(****************************************************************************************)
(*							  Check for valid logical axis no.							*)
(****************************************************************************************)
IF NOT bIsChannelSpecific AND NOT HLI3_CheckAxisValid(nHliAxisIdx := nHliAxisIdx) THEN
	bError									:= TRUE;
	nErrorId								:= 10000;
	RETURN;
END_IF

IF NOT HLI3_CheckChannelValid(nChannel := nHliChannelIdx) THEN
	bError									:= TRUE;
	nErrorId								:= 20000;
	RETURN;	
END_IF

(****************************************************************************************)
(*											Reset										*)
(****************************************************************************************)
fbRtrigChannelReset
	(CLK := bChannelReset);

IF fbRtrigChannelReset.Q THEN
	nRevolution		:= 0;
	nPosition		:= 0;
	bAcknowledge	:= FALSE;
	M03				:= FALSE;
	M03_Internal	:= FALSE;
	M04				:= FALSE;
	M04_Internal	:= FALSE;
	M05				:= FALSE;
	M05_Internal	:= FALSE;
	M19				:= FALSE;
	M19_Internal	:= FALSE;	
	pM40^			:= FALSE;
	M40_Internal	:= FALSE;
	pM41^			:= FALSE;
	M41_Internal	:= FALSE;
	pM42^			:= FALSE;
	M42_Internal	:= FALSE;
	pM43^			:= FALSE;
	M43_Internal	:= FALSE;
	pM44^			:= FALSE;
	M44_Internal	:= FALSE;
	pM45^			:= FALSE;
	M45_Internal	:= FALSE;
END_IF

(****************************************************************************************)
(*									Receive requests from cnc							*)
(****************************************************************************************)
(* Look out for open technology function either on the channel or the axis specific		*)
(* section of the HLI, depending on parameter ''.										*)
IF bIsChannelSpecific THEN
	nOpenTechnoCount	:= gpCh[nHliChannelIdx]^.used_units_std_sync_r;
	nTechFctMaxidx 		:= gpCh[nHliChannelIdx]^.used_units_std_sync_r - 1;
ELSE
	nOpenTechnoCount	:= gpAx[nHliAxisIdx]^.used_units_std_sync_r;
	nTechFctMaxidx 		:= gpAx[nHliAxisIdx]^.used_units_std_sync_r - 1;
END_IF

IF nOpenTechnoCount > 0 THEN
	FOR nLoop := 0 TO nTechFctMaxIdx DO
		(* Depending on the source determined by parameter 'bIsChannelSpecific', the		*)
		(* channel or axis specific section of the HLI will be examined.					*)
		IF bIsChannelSpecific THEN
			pActTechnoUnit	:= ADR(gpCh[nHliChannelIdx]^.techno_unit_std_sync[nLoop]);
		ELSE
			(* Get current axis specifc technology data *)
			pActTechnoUnit	:= ADR(gpAx[nHliAxisIdx]^.techno_unit_std_sync[nLoop]);
		END_IF
	
		(* Check request *)
		IF pActTechnoUnit^.please_rw AND
		   NOT pActTechnoUnit^.done_w
		THEN
			CASE UINT_TO_UDINT(pActTechnoUnit^.fkt_ctrl_r) OF
		     (* -------------------------------------------------------------------------- *)
			 (* Handle M function *)
			 HLI_INTF_M_FKT:
				pMProcess					:= ADR(pActTechnoUnit^.attribut_r.data[0]);
				
				IF (pMProcess > 0) AND bHandleGearChange THEN
					CASE pMProcess^.nr OF
					 40:	M_ManageAcknowledgement(ADR(M40_Internal), pM40, ADR(bAcknowledge));
					 41:	M_ManageAcknowledgement(ADR(M41_Internal), pM41, ADR(bAcknowledge));
					 42:	M_ManageAcknowledgement(ADR(M42_Internal), pM42, ADR(bAcknowledge));
					 43:	M_ManageAcknowledgement(ADR(M43_Internal), pM43, ADR(bAcknowledge));
					 44:	M_ManageAcknowledgement(ADR(M44_Internal), pM44, ADR(bAcknowledge));
					 45:	M_ManageAcknowledgement(ADR(M45_Internal), pM45, ADR(bAcknowledge));
					END_CASE
				END_IF
				
			 (* -------------------------------------------------------------------------- *)
			 (* Handle S function *)
			 HLI_INTF_SPINDEL:
				pSProcess					:= ADR(pActTechnoUnit^.attribut_r.data[0]);
				
				(* If we are working with spindle functions provided by the channel 		*)
				(* specific section of the HLI the logical axis number transmitted from the *)
				(* CNC must fit the one given in parameter 'nLogAxisNoChannelSpecific'!					*)												
				IF bIsChannelSpecific AND (UINT_TO_INT(pSProcess^.log_achs_nr) <> nLogAxisNoChannelSpecific) THEN
					RETURN;
				END_IF
	
				CASE pSProcess^.move_cmd OF
				 (* ----------------------------------------------------------------------- *)
				 0: (* M19 *)
					IF (pSProcess^.pos_cmd = 19) AND
					   NOT M19_Internal THEN
						nPosition			:= pSProcess^.pos;
						M19_Internal		:= TRUE;
						M19					:= TRUE;
					ELSE
						IF NOT M19 THEN
							M19_Internal	:= FALSE;
							bAcknowledge	:= TRUE;
						END_IF
					END_IF
	
				 (* ----------------------------------------------------------------------- *)
				 3: (* M03 *)
					nRevolution				:= pSProcess^.rev;
	
					IF NOT M03_Internal THEN
						M03_Internal		:= TRUE;
						M03					:= TRUE;
					ELSE
						IF NOT M03 THEN
							M03_Internal	:= FALSE;
							bAcknowledge	:= TRUE;
						END_IF
					END_IF
	
				 (* ----------------------------------------------------------------------- *)
				 4: (* M04 *)
					nRevolution				:= pSProcess^.rev;
	
					IF NOT M04_Internal THEN
						M04_Internal		:= TRUE;
						M04					:= TRUE;
					ELSE
						IF NOT M04 THEN
							M04_Internal	:= FALSE;
							bAcknowledge	:= TRUE;
						END_IF
					END_IF
	
				 (* ----------------------------------------------------------------------- *)
				 5: (* M05 *)
					IF NOT M05_Internal THEN
						M05_Internal		:= TRUE;
						M05					:= TRUE;
					ELSE
						IF NOT M05 THEN
							M05_Internal	:= FALSE;
							bAcknowledge	:= TRUE;
						END_IF
					END_IF
	
				END_CASE
			END_CASE
	
			(* Handle acknowledgement *)
			IF bAcknowledge THEN
				bAcknowledge				:= FALSE;
				nRevolution					:= 0;
				nPosition					:= 0;
				pActTechnoUnit^.please_rw 	:= FALSE;
		   		pActTechnoUnit^.done_w		:= TRUE;
			END_IF
		END_IF
	END_FOR
	
END_IF
END_ACTION

{attribute 'object_name' := 'M_ManageAcknowledgement'}
METHOD PRIVATE M_ManageAcknowledgement
VAR_INPUT
	pInternal: POINTER TO BOOL;
	pPublic: POINTER TO BOOL;
	pAcknowledgement: POINTER TO BOOL;
END_VAR
IF NOT pInternal^ THEN
	pInternal^			:= TRUE;
	pPublic^			:= TRUE;	
ELSIF NOT pPublic^ THEN
	pInternal^			:= FALSE;
	pAcknowledgement^	:= TRUE;
END_IF
END_METHOD

END_FUNCTION_BLOCK

// ---- CNC Beckhoff/3 Control/HLI3_SetAxisOverride.TcPOU
FUNCTION HLI3_SetAxisOverride : BOOL
VAR_INPUT
	/// number of Axis 
	nHliAxisIdx: INT;
	nOverride: UINT;
END_VAR

(* ========================================================= *)
(*    FUN: HLI_SetAxisOverride                               *)
(* --------------------------------------------------------- *)
(*   Desc: Set the Axis Override                             *)
(* Author: TV                                                *)
(*   Date: 20.12.2007                                        *)
(*   Rev.: 1.0                                               *)
(*   Rev.: 1.1 MiB 19.11.2012 Tc3                            *)
(* ========================================================= *)
IF NOT (HLI3_CheckAxisValid(nHliAxisIdx := nHliAxisIdx)) THEN
	HLI3_SetAxisOverride := FALSE;
	RETURN;
END_IF


(* Limit the override *)
IF nOverride > 1200	THEN nOverride := 1200; END_IF
IF nOverride < 0 THEN nOverride := 0; END_IF

	gpAx[nHliAxisIdx]^.ipo_mc_control.override.enable_w  := TRUE;
	gpAx[nHliAxisIdx]^.ipo_mc_control.override.command_w := nOverride;

HLI3_SetAxisOverride := TRUE;

END_FUNCTION

// ---- CNC Beckhoff/PRG_ManualMode.TcPOU
PROGRAM PRG_ManualMode
VAR
	
END_VAR

(****************************************************************************************)
(* POU:		PRG_ManualMode                      										*)
(* Type:	PRG																			*)
(* Author: 	HR                                               							*)
(* Date: 	24.01.11																	*)
(* Rev.: 	1.0                                               							*)
(* ------------------------------------------------------------------------------------ *)
(* Desc:	Calls the appropriate manual mode handler									*)
(****************************************************************************************)

(* By default 'geManualModeController' is 'HMI'. Therefore program 'PRG_ManualModeHMI'	*)
(* is called in order to map manual mode signals from HMI to the manual mode control	*)
(* structures. By changing 'geManualModeController´s' value one can call different sub	*)
(* programs to set them in a application specific way.
									*)
geManualModeController := HMI;


CASE geManualModeController OF
	HMI:		PRG_ManualModeHMI();
	PANEL:		;
	REMOTE:		;
	CUSTOMER:	;
END_CASE

END_PROGRAM

// ---- CNC Beckhoff/PRG_ManualModeHMI.TcPOU
PROGRAM PRG_ManualModeHMI
VAR
	fbUintUdInt: ARRAY [0..MAX_USED_CHANNEL_IDX] OF FB_Uint_Udint;
	nHandwheel : UINT;		(* increments for handwheel (e.g. EL5101   *)
	nHandWheelBig: UDINT;
	i: INT;
END_VAR


FOR i := 0 TO MAX_USED_CHANNEL_IDX DO
	
	IF (HLI3_CheckChannelValid(i)) THEN

		stManualModeParameter[i].stChannelParameter.nChanIdx						:= i;       (* Channel 1 *)
		stManualModeParameter[i].stChannelParameter.nInc							:= PLCMachineMode[i+1].ManualMode.nInc * 10;
		
		stManualModeParameter[i].stChannelParameter.eManualType						:= UINT_TO_INT(PLCMachineMode[i+1].ManualMode.nManualTyp);			
		IF (stManualModeParameter[i].stChannelParameter.eManualType = E_CNC_ManualType.Handwheel AND i <> PLCSelectedChannel-1) THEN	(* if in Handwheel mode and the channel is NOT selected -> leave handwheel mode and change to TippMode*)
			stManualModeParameter[i].stChannelParameter.eManualType						:= E_CNC_ManualType.TippMode;
		END_IF		
		
		stManualModeParameter[i].stChannelParameter.nHandwheelResolution			:= UDINT_TO_DINT(PLCMachineMode[i+1].ManualMode.nHwResolution);    (* 0.1 µm /rev (from HMI) *)						
		stManualModeParameter[i].stAxisParameter.stControlUnit[0].nLogAxisNr		:= PLCMachineMode[i+1].ManualMode.nLogAxisNumber;   (* Log. Achs Nummer *)
		IF stManualModeParameter[i].stAxisParameter.stControlUnit[0].nLogAxisNr = 0 THEN
			stManualModeParameter[i].stAxisParameter.stControlUnit[0].nLogAxisNr := gpCh[i]^.bahn_state.coord_r[0].log_achs_nr_r;
			PLCMachineMode[i+1].ManualMode.nLogAxisNumber := gpCh[i]^.bahn_state.coord_r[0].log_achs_nr_r;
		END_IF
		stManualModeParameter[i].stAxisParameter.stControlUnit[0].nSpeed			:= LREAL_TO_UDINT(PLCMachineMode[i+1].ManualMode.nSpeed * 16.666);
		stManualModeControlElements[i].stControlKeys[0].bKeyNeg						:= PLCMachineMode[i+1].ManualMode.bKeyNeg;
		stManualModeControlElements[i].stControlKeys[0].bKeyPos						:= PLCMachineMode[i+1].ManualMode.bKeyPos;
		stManualModeControlElements[i].stControlKeys[0].bKeyRapid					:= PLCMachineMode[i+1].ManualMode.bKeyRapid;
		
		(* the cnc needs an UDINT for handwheel increments, fbUintUdint extends an UInt to an UDINT *)
		(* the resoltion of the handwheel is parameterized in CNC-Task GEO/Manual MDS: (e.g. 400 handwheel inc / handwheel revolution
		
				hr_data[0].hr_aufl_z              400         ( P-MANU-00005 : Handwheel resolution numerator
				hr_data[0].hr_aufl_n                1     	  ( P-MANU-00006 : Handwheel resolution denominator
		*) 
		fbUintUdInt[i](nInSmall := nHandwheel, nBig := nHandWheelBig);
		stManualModeControlElements[i].nHandwheelInc[0] :=  UDINT_TO_DINT(nHandWheelBig);
  END_IF
END_FOR

END_PROGRAM

// ---- CNC Beckhoff/Util/FB_Uint_Udint.TcPOU
FUNCTION_BLOCK FB_Uint_Udint
VAR
	nOldValue: UINT;
	nDiff: DINT;
	nMinus: BOOL;
	nPlus: BOOL;
END_VAR
VAR_INPUT
	nInSmall: UINT;
END_VAR

VAR_IN_OUT
	nBig: UDINT;
END_VAR

nDiff := nInSmall - nOldValue;


(* Richtung Minus *)
IF ndiff > 10000 THEN
	nBig := nBig - 1;
	nMinus := TRUE;
END_IF

(* Richtung Plus *)
IF ndiff < -10000 THEN
	nBig := nBig + 1;
	nPlus := TRUE;
END_IF

IF (ndiff < 500) AND ndiff > -500 THEN
  nBig := DINT_TO_UDINT( UDINT_TO_DINT(nBig) + nDiff) ;
END_IF
nOldValue := nInSmall;

END_FUNCTION_BLOCK

// ---- CNC Beckhoff/PRG_ChannelHandler.TcPOU
PROGRAM PRG_ChannelHandler
VAR	
	nChan					: INT;
	nOldSelectedChannel		: UDINT;
	CNCChannel				: ARRAY[0..MAX_USED_CHANNEL_IDX] OF HLI3_CNCChannel;	
	BlockSearch_Channel		: ARRAY[0..MAX_USED_CHANNEL_IDX] OF HLI3_BlockSearch;
	ModeManual_Channel		: ARRAY[0..MAX_USED_CHANNEL_IDX] OF HLI3_ManualModeHandler;
	ErrorHandler_Channel	: ARRAY[0..MAX_USED_CHANNEL_IDX] OF FB_ChannelError;
	nChanNo: UDINT;	
	i: INT;
	
END_VAR

(****************************************************************************************)
(* POU:		PRG_ChannelHandler                     										*)
(* Type:	PRG																			*)
(* Author: 	HR / TV / MiB                                          						*)
(* Date: 	23.01.11																	*)
(* Last:	02.03.16																	*)
(* Rev.: 	1.4                                              							*)
(* ------------------------------------------------------------------------------------ *)
(* Desc:	Description																	*)
(****************************************************************************************)

(****************************************************************************************)
(*	  Map CNC function selection from HMI to selected channel (and state vice versa)  	*)
(****************************************************************************************)
IF (nOldSelectedChannel <>INT_TO_UDINT(PLCSelectedChannel)) THEN
	PLCChannelSignals.SingleBlock 		:= PLCMachineMode[PLCSelectedChannel].ChannelSignals.SingleBlock;
	PLCChannelSignals.PrgBlockIgnore	:= PLCMachineMode[PLCSelectedChannel].ChannelSignals.PrgBlockIgnore;
	PLCChannelSignals.M01Stop 			:= PLCMachineMode[PLCSelectedChannel].ChannelSignals.M01Stop;
	PLCChannelSignals.Backward 			:= PLCMachineMode[PLCSelectedChannel].ChannelSignals.Backward;
	PLCChannelSignals.FeedHold 			:= PLCMachineMode[PLCSelectedChannel].ChannelSignals.FeedHold;
	nOldSelectedChannel 				:= INT_TO_UDINT(PLCSelectedChannel);
END_IF

PLCMachineMode[PLCSelectedChannel].ChannelSignals.SingleBlock 		:= PLCChannelSignals.SingleBlock;
PLCMachineMode[PLCSelectedChannel].ChannelSignals.PrgBlockIgnore 	:= PLCChannelSignals.PrgBlockIgnore;
PLCMachineMode[PLCSelectedChannel].ChannelSignals.M01Stop 			:= PLCChannelSignals.M01Stop;
PLCMachineMode[PLCSelectedChannel].ChannelSignals.Backward 		:= PLCChannelSignals.Backward;
PLCMachineMode[PLCSelectedChannel].ChannelSignals.FeedHold 		:= PLCChannelSignals.FeedHold;



FOR i := 0 TO MAX_USED_CHANNEL_IDX DO
		
	nChan := i;	
	IF (HLI3_CheckChannelValid(nChan)) THEN		
		
		(* Error handler for channel 1 *)
		ErrorHandler_Channel[nChan](nChanIdx			:= nCHan);
		
		(* Pass feedrate override from HMI to first channel (in [0.1%]) *)
		HLI3_SetChannelOverride
			(nChanIdx			:= nChan,
			 nOverride			:= PLCFeedOverride * 10
			);
		
		(* Channel interface *)
		CNCChannel[nChan]
			(nChanIdx			:= nChan,
			 (* Operation Mode *)
			 bModeStandby		:= PLCMachineMode[nChan+1].Standby,
			 bModeAutomatic		:= PLCMachineMode[nChan+1].Automatic,
			 bModeManual		:= PLCMachineMode[nChan+1].Manual,
			 bModeMDI			:= PLCMachineMode[nChan+1].MDI,	 
			 bModeReference		:= PLCMachineMode[nChan+1].Homing,
			 (* Operation State *)
			 bStateSelect		:= PLCMachineMode[nChan+1].Select,
			 bStateReady		:= PLCMachineMode[nChan+1].Ready,
			 bStateStart		:= PLCMachineMode[nChan+1].Start,
			 bStateStop			:= PLCMachineMode[nChan+1].Stop,
			 bStateReset		:= PLCMachineMode[nChan+1].Reset,
			 (* Special Functions *)
			 sProgramName		:= PLCMachineMode[nChan+1].ProgramName,
			 sMDIString			:= PLCMachineMode[nChan+1].MDIString,
			 bBackwardMotion	:= PLCMachineMode[nChan+1].ChannelSignals.Backward,
			 bPrgBlockIgnore	:= PLCMachineMode[nChan+1].ChannelSignals.PrgBlockIgnore,
			 bFeedHold			:= PLCMachineMode[nChan+1].ChannelSignals.FeedHold,
			 bSingleBlock		:= PLCMachineMode[nChan+1].ChannelSignals.SingleBlock,
			 bDoSingleBlock		:= PLCMachineMode[nChan+1].ChannelSignals.DoSingleBlock,
			 bM01Stop			:= PLCMachineMode[nChan+1].ChannelSignals.M01Stop,
			 nSyntaxCheck		:= PLCMachineMode[nChan+1].SyntaxCheck.nType,
			 sManualInitString  :=  stManualModeParameter[nChan].stChannelParameter.strInitParameter
			);
		
		(* Handle block search *)
		BlockSearch_Channel[nChan]
			(nChanIdx			:= nChan,
			 bStartRead      	:= PLCMachineMode[nChan+1].BlockSearch.bStartRead,   (* Edge signal *)
			 bStartWrite     	:= PLCMachineMode[nChan+1].BlockSearch.bStartWrite,  (* Edge signal *)
			 BlockSearch		:= PLCMachineMode[nChan+1].BlockSearch
			);
		
		CNCSystem.Channel[nChan].ActDistance 	:= DINT_TO_LREAL(BlockSearch_Channel[nChan].coveredDistance_AfterReset) / 10.0;
		CNCSystem.Channel[nChan].ActBlockCount 	:= BlockSearch_Channel[nChan].actualBlockCount_AfterReset;
		
		
		ModeManual_Channel[nChan]
			(stManualModeParameter  	 	:= stManualModeParameter[nChan],
			 stManualModeControlElements	:= stManualModeControlElements[nChan],
			 stManualModeControlElementState := stManualModeControlElementState,
			 bReset 						:= FALSE,
			 arrAxisInG201 				=> stManualModeState[nChan].arrAxisInG201
			);
	END_IF
END_FOR

END_PROGRAM

// ---- CNC Beckhoff/2 OperationMode/HLI3_CNCChannel.TcPOU
FUNCTION_BLOCK HLI3_CNCChannel
VAR_INPUT
	/// index of channel 
	nChanIdx: INT;
	/// must be xxx.nc 
	sProgramName: STRING(HLI_IMCM_MODE_STATE_PARAM_STRL);
	/// the MDI string 
	sMDIString: STRING(HLI_IMCM_MODE_STATE_PARAM_STRL);
	/// static signal 
	bBackwardMotion: BOOL;
	/// static signal 
	bFeedHold: BOOL;
	/// static signal 
	bReducedFeed: BOOL;
	/// static signal 
	bSingleBlock: BOOL;
	/// static signal 
	bPrgBlockIgnore: BOOL;
	/// static signal 
	bM01Stop: BOOL;
	/// static signal 
	nSyntaxCheck: DINT;
	/// initi parameter for manual mode
	sManualInitString	     : STRING;
END_VAR
VAR_IN_OUT
	/// please only a flank 
	bModeStandby: BOOL;
	/// please only a flank 
	bModeAutomatic: BOOL;
	/// please only a flank 
	bModeManual: BOOL;
	/// please only a flank 
	bModeMDI: BOOL;
	/// please only a flank 
	bModeReference: BOOL;
	/// please only a flank 
	bStateSelect: BOOL;
	/// please only a flank 
	bStateReady: BOOL;
	/// please only a flank 
	bStateStart: BOOL;
	/// please only a flank 
	bStateStop: BOOL;
	/// please only a flank 
	bStateReset: BOOL;
	/// please only a flank 
	bDoSingleBlock: BOOL;
END_VAR
VAR
	bGoToActive	: BOOL;
	/// Pointer to HLI Motion Control Unit 
	pUnit: POINTER TO MC_CONTROL_MCM_MODE_STATE_UNIT;
	/// Pointer to HLI channel command 
	pCommand: POINTER TO HLI_PROC_TRANS_TO_MODE_STATE;
	/// Pointer to channel control structure 
	pChannel: POINTER TO ST_CncChannel;
	ChannelMHTFunction: HLI3_QuitChannelMHTFunction;
	/// Current Mode of Operation Modes;
	currentMode: UDINT;
	/// Current State of Operation Modes;
	currentState: UDINT;
	idx: INT;
	bEndOfManualMode: BOOL;
	bCheckOpModeFirst: BOOL;
	fbRTrigReset: R_TRIG;
	bResetRequest: BOOL;
	ChannelResetRequest: HLI3_ChannelResetRequest;
	nChan: INT;
	nStateAutoMDIStart: INT;
END_VAR

(* ========================================================= *)
(*     FB: HLI_CNCChannel                                    *)
(* --------------------------------------------------------- *)
(*   Desc:                                                   *)
(*   Author: MK ,MiB, TV, Rch                                *)
(*   Date: 2017.05.08                                        *)
(*   Rev.: 1.6                                               *)
(*         1.2 Before "start" the state is swicthed to 		 *)
(*				"Selected" and "Ready" to ensure that the    *)	
(*				actual selected program will start 			 *)
(*		   1.3  BugFix : nChanNo at HLI3_ChannelModeMDI()    *)
(*         1.4  Implement state switch to "selected" and "ready"  *)         
(*		   1.5  Channel reset via commanding state 			 *)
(*              RESETTING directly							 *)  
(*		   1.6  Optimized Channel reset via commanding state *)
(*				RESETTING directly						     *)
(*		   1.7  Init Paramerer for Manual mode as input parameter*)
(* ========================================================= *)

IF NOT HLI3_CheckChannelValid(nChannel := nChanIdx) THEN
	RETURN;
END_IF


(* handle reset request *)
fbRTrigReset
	(CLK := bStateReset);
	
IF fbRTrigReset.Q THEN
	nStateAutoMDIStart := 0;
END_IF

(* set up pointer *)
pUnit    := ADR(gpCh[nChanIdx]^.channel_mc_control.mode_and_state);
pCommand := ADR(pUnit^.command_w);


(* ************************************* *)
(*  Motion-Control                       *)
(* ************************************* *)
(* Backward Motion *)
HLI3_ChannelSetBackwardMotion(nChanIdx:=nChanIdx, bBackwardMotion:=bBackwardMotion);

(* Program Block Ignore *)
HLI3_ChannelSetProgramBlockIgnore(nChanIdx:=nChanIdx, bPrgBlockIgnore:=bPrgBlockIgnore);

(* Feed Hold *)
HLI3_ChannelSetFeedHold(nChanIdx:=nChanIdx, bFeedHold:=bFeedHold);

(* Single Step *)
HLI3_ChannelSetSingleBlock(nChanIdx:=nChanIdx, bSingleBlock:=bSingleBlock);

(* Reduced Feed *)
HLI3_ChannelSetReducedFeed(nChanIdx:=nChanIdx, bReducedFeed:=bReducedFeed);

(* Syntax Check *)
gpCh[nChanIdx]^.decoder_mc_control.execution_mode.command_w := nSyntaxCheck;

(* Optional stop M01 *)
gpCh[nChanIdx]^.bahn_mc_control.m01_stop_enable.command_w := bM01Stop;


(* ************************************ *)
(*  MHT-Function                        *)
(* ************************************ *)
(* Reset all M- and H-Functions whenn 	*)
(* the channel gets resetted			*)
IF (pChannel > 0) THEN
	IF (pChannel^.ActState = HLI_IMCM_PROCESS_RESETTING) THEN
		HLI3_ChannelResetMFunctions(nChanIdx);
		HLI3_ChannelResetHFunctions(nChanIdx);
	END_IF
END_IF

(* MHT-Function, channel *)
ChannelMHTFunction(nChanIdx:=nChanIdx);

(* ************************************* *)
(*  Channel Status Info and error        *)
(* ************************************* *)
HLI3_GetChannelStatusInfo(nChanIdx:=nChanIdx);
HLI3_GetChannelError(nChanIdx:=nChanIdx);

(* ************************************* *)
(*  do single stepping                   *)
(* ************************************* *)
(* Achtung: hier noch anpassen, nur in Abhaengigkeit vom aktuellen Status den Start setzen *)
IF bDoSingleBlock THEN
	bDoSingleBlock := FALSE;
	bStateStart 	:= TRUE;
END_IF

(* ************************************* *)
(*  Operation Modes                      *)
(* ************************************* *)
(* Target modes and states *)
pChannel := ADR(CNCSystem.Channel[nChanIdx]);
OpModes();

(* OperationMode Standby *)
IF pChannel^.Mode.Standby = TRUE THEN
	HLI3_ChannelModeStandby(ProgramName:=sProgramName, pUnit:=pUnit, pCommand:=pCommand, pChannel:=pChannel);
END_IF

(* OperationMode Auto *)
IF pChannel^.Mode.Auto = TRUE THEN
	HLI3_ChannelModeAuto(ProgramName:=sProgramName, pUnit:=pUnit, pCommand:=pCommand, pChannel:=pChannel);
END_IF

(* OperationMode MDI *)
IF pChannel^.Mode.MDI THEN
	(*sProgramName := PLCCncMDIString;*)
	HLI3_ChannelModeMDI(pMDIString:=ADR(sMDIString), pUnit:=pUnit, pCommand:=pCommand, pChannel:=pChannel);
END_IF

(* OperationMode Reference *)
//IF pChannel^.Mode.REFERENCE THEN TC3HR
IF pChannel^.Mode.Homing THEN
	sProgramName := '';	(* we choose the default program: rpf.nc *)
	HLI3_ChannelModeReference(sRefPosString:=sProgramName, pUnit:=pUnit, pCommand:=pCommand, pChannel:=pChannel);
END_IF

(* OperationMode Manual *)
IF pChannel^.Mode.Manual THEN
	bEndOfManualMode := FALSE;
	HLI3_ChannelModeManual(pUnit:=pUnit, pCommand:=pCommand, pChannel:=pChannel, sManualInitString := sManualInitString);
END_IF

(* end of manual mode *)
IF (pChannel^.Mode.Standby
OR pChannel^.Mode.Auto
OR pChannel^.Mode.MDI
//OR pChannel^.Mode.REFERENCE) THEN TC3HR
OR pChannel^.Mode.Homing) THEN
	bEndOfManualMode := TRUE;
END_IF

(* Reset *)
HLI3_ChannelReset(nChanIdx:=nChanIdx);							(* channel *)
FOR idx := 0 TO UDINT_TO_INT(gNrAx) DO							(* axis *)
	HLI3_AxisReset(nChanNo:=nChanIdx+1, nHliAxisIdx:=idx);
END_FOR

ACTION AutoMDIStart:



CASE nStateAutoMDIStart OF
	0:		;(* IDLE *)
	
	10: (* swicth to selected *)
		pChannel^.State.Selected := TRUE;
		nStateAutoMDIStart := nStateAutoMDIStart +10;
		
	20: (* wait for selected *)
		IF (pChannel^.ActState =  HLI_IMCM_PROCESS_SELECTED) THEN
			pChannel^.State.Ready := TRUE;
			nStateAutoMDIStart := nStateAutoMDIStart +10;
		END_IF
	30: (* Wait for ready and then start*)
		IF (pChannel^.ActState =  HLI_IMCM_PROCESS_READY) THEN
			pChannel^.State.Start := TRUE; 
			nStateAutoMDIStart := 0;
		END_IF
	
END_CASE
END_ACTION

ACTION OpModes:
(*************************************************)
(* Restore internal state at first run           *)
(* after PLC reset                               *)
(*************************************************)

IF bCheckOpModeFirst = FALSE THEN
	bCheckOpModeFirst := TRUE;
	currentMode := HLI3_GetChannelMode(nChanIdx:=nChanIdx);
	IF currentMode = HLI_IMCM_STANDBY_MODE THEN
		pChannel^.Mode.Standby := TRUE;
	END_IF
	IF currentMode = HLI_IMCM_AUTOMATIC_MODE THEN
		pChannel^.Mode.Auto := TRUE;
	END_IF
	IF currentMode = HLI_IMCM_MDI_MODE THEN
		pChannel^.Mode.MDI := TRUE;
	END_IF
	IF currentMode = HLI_IMCM_MANUAL_MODE THEN
		pChannel^.Mode.Manual := TRUE;
	END_IF
	IF currentMode = HLI_IMCM_REFERENCE_MODE THEN
		//pChannel^.Mode.REFERENCE := TRUE; TC3HR
		pChannel^.Mode.Homing := TRUE;
	END_IF
END_IF


(*************************************************)
(* Operation Modes                               *)
(*************************************************)

IF bModeStandby THEN
	bModeStandby := FALSE;
	pChannel^.Mode.Standby		:= TRUE;
	pChannel^.Mode.Auto			:= FALSE;
	pChannel^.Mode.MDI			:= FALSE;
	pChannel^.Mode.Manual		:= FALSE;
	pChannel^.Mode.Homing		:= FALSE;


	pChannel^.State.Selected	:= TRUE;
END_IF

IF bModeAutomatic THEN
	bModeAutomatic 				:= FALSE;
	bGoToActive					:= FALSE;
	pChannel^.Mode.Standby		:= FALSE;
	pChannel^.Mode.Auto			:= TRUE;
	pChannel^.Mode.MDI			:= FALSE;
	pChannel^.Mode.Manual		:= FALSE;
	pChannel^.Mode.Homing		:= FALSE;

	pChannel^.State.Selected	:= TRUE;
END_IF

IF bModeMDI THEN
	bModeMDI := FALSE;
	bGoToActive					:= FALSE;
	pChannel^.Mode.Standby		:= FALSE;
	pChannel^.Mode.Auto			:= FALSE;
	pChannel^.Mode.MDI			:= TRUE;
	pChannel^.Mode.Manual		:= FALSE;
	pChannel^.Mode.Homing		:= FALSE;

	pChannel^.State.Selected	:= TRUE;
END_IF

IF bModeManual THEN
	bModeManual := FALSE;
	pChannel^.Mode.Standby		:= FALSE;
	pChannel^.Mode.Auto			:= FALSE;
	pChannel^.Mode.MDI			:= FALSE;
	pChannel^.Mode.Manual		:= TRUE;
	pChannel^.Mode.Homing		:= FALSE;

	pChannel^.State.Start		:= TRUE;
END_IF

IF bModeReference THEN
	bModeReference := FALSE;
	bGoToActive					:= FALSE;
	pChannel^.Mode.Standby		:= FALSE;
	pChannel^.Mode.Auto			:= FALSE;
	pChannel^.Mode.MDI			:= FALSE;
	pChannel^.Mode.Manual		:= FALSE;
	pChannel^.Mode.Homing		:= TRUE;
	
	pChannel^.State.Start		:= TRUE;
END_IF



(*************************************************)
(* Operation States                              *)
(*************************************************)

currentMode := HLI3_GetChannelMode(nChanIdx:=nChanIdx);
currentState := HLI3_GetChannelState(nChanIdx:=nChanIdx);

CASE currentMode OF
	(*-------------------------------------------------------------------*)
	HLI_IMCM_STANDBY_MODE:
		IF bStateReset THEN
			pChannel^.Mode.Standby := TRUE;
			pChannel^.State.Reset := TRUE;
		END_IF

	(*-------------------------------------------------------------------*)
	HLI_IMCM_AUTOMATIC_MODE:
		IF bStateStart THEN  (* replaced a simple 'start' by a sequence which switches the state to selected and ready*)
			IF currentState <> HLI_IMCM_PROCESS_HOLD AND currentState <> HLI_IMCM_PROCESS_ACTIVE THEN
				nStateAutoMDIStart := 10;
			ELSE
				pChannel^.State.Start := TRUE; 
			END_IF					   	
		END_IF
		IF nStateAutoMDIStart <> 0 THEN
			AutoMDIStart();
		END_IF

		IF bStateStop AND currentState <> HLI_IMCM_PROCESS_DESELECTED THEN
			pChannel^.State.Stop := TRUE;
		END_IF

		IF bStateReady THEN
			pChannel^.State.Ready := TRUE;
		END_IF

		IF bStateReset THEN
			pChannel^.State.Reset := TRUE;
		END_IF
		
		IF bStateSelect THEN
			pChannel^.State.Selected := TRUE;
		END_IF		

	(*-------------------------------------------------------------------*)
	HLI_IMCM_MDI_MODE:
		IF bStateStart THEN
			IF currentState <> HLI_IMCM_PROCESS_HOLD AND currentState <> HLI_IMCM_PROCESS_ACTIVE THEN
				nStateAutoMDIStart := 10;
			ELSE
				pChannel^.State.Start := TRUE; 
			END_IF
		END_IF
		
		IF nStateAutoMDIStart <> 0 THEN
			AutoMDIStart();
		END_IF
		
		IF bStateStop AND currentState <> HLI_IMCM_PROCESS_DESELECTED THEN
			pChannel^.State.Stop := TRUE;
		END_IF

		IF bStateSelect THEN
			pChannel^.State.Selected := TRUE;
		END_IF
		
		IF bStateReady THEN
			pChannel^.State.Ready := TRUE;
		END_IF

		IF bStateReset THEN
			pChannel^.State.Reset := TRUE;
		END_IF

	(*-------------------------------------------------------------------*)
	HLI_IMCM_MANUAL_MODE:
		IF bStateStart OR ((currentState = HLI_IMCM_PROCESS_SELECTED) AND bGoToActive) THEN
			pChannel^.State.Start 	:= TRUE;
		END_IF

		IF bStateReady THEN
			pChannel^.State.Ready 	:= TRUE;
		END_IF

		IF bStateSelect THEN
			pChannel^.State.Selected := TRUE;
		END_IF

		IF bStateStop THEN
			pChannel^.State.Stop := TRUE;
		END_IF

		IF bStateReset THEN
			bGoToActive := TRUE;
			pChannel^.State.Reset := TRUE;
		END_IF

	(*-------------------------------------------------------------------*)
	HLI_IMCM_REFERENCE_MODE:
		IF bStateStart THEN
			pChannel^.State.Start := TRUE;
		END_IF

		IF bStateStop THEN
			pChannel^.State.Stop := TRUE;
		END_IF

		IF bStateReset THEN
			pChannel^.State.Reset := TRUE;
		END_IF
END_CASE


bStateStart 	:= FALSE;
bStateStop 		:= FALSE;
bStateReset 	:= FALSE;
bStateSelect 	:= FALSE;
bStateready 	:= FALSE;
END_ACTION

END_FUNCTION_BLOCK

// ---- CNC Beckhoff/4 MHT-Function/HLI3_QuitChannelMHTFunction.TcPOU
FUNCTION_BLOCK HLI3_QuitChannelMHTFunction
VAR_INPUT
	/// Number of channel 
	nChanIdx: INT;
END_VAR
VAR_OUTPUT
	bOK: BOOL;
END_VAR
VAR
	ChannelMFunction: HLI3_DoChannelMFunction;
	ChannelTFunction: HLI3_DoChannelTFunction;
	ChannelHFunction: HLI3_DoChannelHFunction;
	/// local pointer to Data of actual Channel 
	pChannelData: POINTER TO HIGH_LEVEL_INTERFACE_CH;
	/// local pointer to actual techno unit 
	pActTechnoUnit: POINTER TO TECHNO_UNIT_CH;
	/// Index of axis specific technology function at HLI 
	nTechFctMaxIdx: UINT;
	/// loop variable 
	idx: UINT;
	/// number of M-function 
	nFuncNr: UDINT;
	nArgument: DINT;
	/// basis id of a tool 
	nToolBasicId: UDINT;
	pMHProcess: POINTER TO HLI_M_H_PROZESS;
	pSProcess: POINTER TO HLI_S_PROZESS;
	pTProcess: POINTER TO HLI_T_PROZESS;
	stAttributeData: St_TechnoAttributeData;
END_VAR

(* ========================================================= *)
(*     FB: HLI3_QuitChannelMHTFunction                        *)
(* --------------------------------------------------------- *)
(*   Desc:                                                   *)
(* Author: MK                                                *)
(*   Rev.: 1.1                                               *)
(*   Date: 18.07.2002                                        *)
(*       : 08.04.2005                                        *)
(*          24.11.2010 MiB Erweiterung um H Funktionen 		 *)
(* ========================================================= *)
(* Rev.:	1.2												 *)
(* Date:	02.10.2010                                    	 *)
(* Author:	HR												 *)
(* Author:	Added support for additional m function number	 *)
(* ========================================================= *)
(* Rev.:	1.3												 *)
(* Date:	26.01.2011                                    	 *)
(* Author:	HR												 *)
(* Author:	Added support for additional h function number	 *)
(* ========================================================= *)
(* Rev.:	1.4												 *)
(* Date:	20.11.2012                                    	 *)
(* Author:	MiB												 *)
(* Author:	TC3												 *)
(* ========================================================= *)
(* Rev.:	1.4.1									         *)
(* Date:	15.07.2013                                    	 *)
(* Author:	TV												 *)
(* ========================================================= *)

IF NOT HLI3_CheckChannelValid(nChannel := nChanIdx) THEN
	bOK := FALSE;
	RETURN; (* A b b r u c h *)
END_IF


(* get pointer to channel data *)
pChannelData := gpCh[nChanIdx];

pActTechnoUnit := ADR(pChannelData^.techno_unit_std_sync[0]);

(* test if there are open synchronisations  *)
IF pChannelData^.used_units_std_sync_r > 0 THEN

	nTechFctMaxIdx := pChannelData^.used_units_std_sync_r - 1;

	FOR idx := 0 TO nTechFctMaxIdx DO
		(* get pointer to actual techno unit *)
		pActTechnoUnit := ADR(pChannelData^.techno_unit_std_sync[idx]);
	
	
		(* test if this M-function has to be acknowledged *)
		IF pActTechnoUnit^.please_rw = TRUE AND				(* request from CNC *)
		   pActTechnoUnit^.done_w = FALSE AND				(* not acknowledged *)
		   pActTechnoUnit^.fkt_ctrl_r = HLI_INTF_M_FKT		(* M-function *)
		THEN
			(* Read number of M-function *)
			pMHProcess := ADR(pActTechnoUnit^.attribut_r.data[0]);
			nFuncNr    := pMHProcess^.nr;
			nArgument	:= pMHProcess^.add_nr_r;
			
			
			stAttributeData.nFunctionNumber_r := pMHProcess^.nr;
			stAttributeData.nTime_r		:= pMHProcess^.zeit;
			stAttributeData.nArgument_r 		:= pMHProcess^.add_nr_r;
			stAttributeData.nBlockNumber_r 	:= pMHProcess^.satz_nr;
			stAttributeData.nPrgLineNumber_r	:= pMHProcess^.prg_zeilen_nr;
			
	
			ChannelMFunction(nChanIdx:=nChanIdx, stTechnoAttributeData := stAttributeData);
			IF ChannelMFunction.bBusy = FALSE THEN
				(* acknowledge this M-function *)
				pActTechnoUnit^.please_rw := FALSE;
				pActTechnoUnit^.done_w := TRUE;
				ADSLOG(strMsg:='acknowledge of M-function: %d', nDINT:=UDINT_TO_DINT(nFuncNr), strArg:='');
			END_IF
	
			bOK := TRUE;
		END_IF


		(* test if this H-function has to be acknowledged *)
		IF pActTechnoUnit^.please_rw = TRUE AND						(* request from CNC *)
		   pActTechnoUnit^.done_w = FALSE AND						(* not acknowledged *)
		   pActTechnoUnit^.fkt_ctrl_r = HLI_INTF_H_FKT		(* H-function *)
		THEN
			(* Read number of H-function *)
			pMHProcess := ADR(pActTechnoUnit^.attribut_r.data[0]);
			stAttributeData.nFunctionNumber_r := pMHProcess^.nr;
			stAttributeData.nTime_r		:= pMHProcess^.zeit;
			stAttributeData.nArgument_r 		:= pMHProcess^.add_nr_r;
			stAttributeData.nBlockNumber_r 	:= pMHProcess^.satz_nr;
			stAttributeData.nPrgLineNumber_r	:= pMHProcess^.prg_zeilen_nr;
	
			ChannelHFunction(nChanIdx:=nChanIdx, stTechnoAttributeData:= stAttributeData);

			(* acknowledge this H-function *)
			IF ChannelHFunction.bBusy = FALSE THEN
					(* acknowledge this H-function *)
				pActTechnoUnit^.please_rw := FALSE;
				pActTechnoUnit^.done_w := TRUE;
				ADSLOG(strMsg:='acknowledge of H-function: %d', nDINT:=UDINT_TO_DINT(nFuncNr), strArg:='');
			END_IF
			bOK := TRUE;
		END_IF
	
		(* test if this T-function has to be acknowledged *)
		IF pActTechnoUnit^.please_rw = TRUE AND				(* request from CNC *)
		   pActTechnoUnit^.done_w = FALSE AND				(* not acknowledged *)
		   pActTechnoUnit^.fkt_ctrl_r = HLI_INTF_TOOL		(* T-function *)
		THEN
			(* Read number of T-function *)
			pTProcess    := ADR(pActTechnoUnit^.attribut_r.data[0]);
			nToolBasicId := DINT_TO_UDINT(pTProcess^.id.basic);
	
			ChannelTFunction(nChanIdx:=nChanIdx, nFuncNr:=nToolBasicId);
	
			(* acknowledge this T-function *)
			pActTechnoUnit^.please_rw := FALSE;
			pActTechnoUnit^.done_w := TRUE;
			ADSLOG(strMsg:='acknowledge of T-function: %d', nDINT:=UDINT_TO_DINT(nToolBasicId), strArg:='');
	
			bOK := TRUE;
		END_IF
	
	END_FOR

END_IF


(*
	HLI_INTF_H_FKT                 :    INT:=2;
	HLI_INTF_SPINDEL              :    INT:=3;
	HLI_INTF_TOOL                 :    INT:=4;
	GCW_250_HLIIntfAxBlock              :    INT:=5;
	GCW_250_HLIIntfVEVariable           :    INT:=6;
	GCW_250_HLIIntfVEVariable_1         :    INT:=7;
	GCW_250_HLIIntfVEVariable_2         :    INT:=8;
	GCW_250_HLIIntfUnknown              :    INT:=9;
*)

(*******************************************************************************************************************)

FOR idx := 0 TO INT_TO_UINT(HLI_TU_CH_LATE_SYNC_MAXIDX) DO
	IF pChannelData^.techno_unit_late_sync[idx].please_rw = TRUE
	AND pChannelData^.techno_unit_late_sync[idx].done_w = FALSE THEN

		(* get pointer to actual techno unit *)
		pActTechnoUnit := ADR(pChannelData^.techno_unit_late_sync[idx]);

		IF pActTechnoUnit^.please_rw = TRUE AND				(* request from CNC *)
			pActTechnoUnit^.done_w = FALSE AND				(* not acknowledged *)
			pActTechnoUnit^.fkt_ctrl_r = HLI_INTF_M_FKT		(* M-function *)
		THEN
			pMHProcess := ADR(pActTechnoUnit^.attribut_r.data[0]);
			nFuncNr    := pMHProcess^.nr;
			
			stAttributeData.nFunctionNumber_r := pMHProcess^.nr;
			stAttributeData.nTime_r		:= pMHProcess^.zeit;
			stAttributeData.nArgument_r 		:= pMHProcess^.add_nr_r;
			stAttributeData.nBlockNumber_r 	:= pMHProcess^.satz_nr;
			stAttributeData.nPrgLineNumber_r	:= pMHProcess^.prg_zeilen_nr;

			ChannelMFunction(nChanIdx:=nChanIdx, stTechnoAttributeData:=stAttributeData);
			IF ChannelMFunction.bBusy = FALSE THEN
			(* acknowledge this M-function *)
			pActTechnoUnit^.please_rw := FALSE;
			pActTechnoUnit^.done_w := TRUE;
			ADSLOG(strMsg:='acknowledge of M-function: %d', nDINT:=UDINT_TO_DINT(nFuncNr), strArg:='');
			(* ADSLOGDINT( msgCtrlMask := ADSLOG_MSGTYPE_MSGBOX OR
										ADSLOG_MSGTYPE_LOG,
						msgFmtStr := 'Channel acknowledge of M-function: %d',
						dintArg := pMHProcess^.nr);
			*)
		END_IF
		bOK := TRUE;

	(*	ELSIF   pActTechnoUnit^.fkt_ctrl_r = HLI_INTF_SPINDEL THEN (* spindle-function *)

 			(* Example: read number of S-function *)
			pSProzess := ADR(pActTechnoUnit^.attribut_r.data[0]);
			ADSLOGDINT( msgCtrlMask := ADSLOG_MSGTYPE_MSGBOX OR
										ADSLOG_MSGTYPE_LOG,
						msgFmtStr := 'Late synch : %d',
						dintArg := pSProzess^.move_cmd);

		ELSIF   pActTechnoUnit^.fkt_ctrl_r = HLI_INTF_TOOL THEN

			pHLI_T_PROZESS := ADR(pActTechnoUnit^.attribut_r.data[0]);
			ADSLOGDINT( msgCtrlMask := ADSLOG_MSGTYPE_MSGBOX OR
										ADSLOG_MSGTYPE_LOG,
						msgFmtStr := 'Late tool process: %d',
						dintArg := pTProcess^.id.basic);*)
		(*ELSE
				ADSLOGDINT( msgCtrlMask := ADSLOG_MSGTYPE_MSGBOX OR
											ADSLOG_MSGTYPE_LOG,
							msgFmtStr := 'Channel acknowledge unknown type: %d',
							dintArg := pActTechnoUnit^.fkt_ctrl_r);*)
		END_IF

	END_IF
END_FOR
(**********************************************************************************************************************)

END_FUNCTION_BLOCK

// ---- CNC Beckhoff/4 MHT-Function/HLI3_DoChannelMFunction.TcPOU
FUNCTION_BLOCK HLI3_DoChannelMFunction
VAR_INPUT
	/// Channel number 
	nChanIdx: INT;
	stTechnoAttributeData: St_TechnoAttributeData;
END_VAR
VAR_OUTPUT
	bBusy: BOOL;
END_VAR
VAR
	pChannel: POINTER TO ST_CncChannel;
END_VAR

(* ========================================================= *)
(*     FB: HLI_DoChannelMFunction                            *)
(* --------------------------------------------------------- *)
(*   Desc:                                                   *)
(* Author: MK                                                *)
(*   Rev.: 1.1                                               *)
(*   Date: 18.07.2002                                        *)
(*       : 08.04.2005                                        *)
(* ========================================================= *)
(* Rev.:	1.2												 *)
(* Date:	02.10.2010                                   	 *)
(* Author:	HR												 *)
(* Author:	Added support for additional m function number	 *)
(*			via new input variable 'nArg'				 	 *)
(* ========================================================= *)
(* Rev.:	1.3												 *)
(* Date:	23.11.2012                                   	 *)
(* Author:	TV, MiB											 *)
(* Author:	structure St_TechnoAttributeData instead of      *)
(*			simple bool array	 							 *)
(* ========================================================= *)

bBusy := TRUE;
IF NOT HLI3_CheckChannelValid(nChannel := nChanIdx) THEN
	RETURN; (* A b b r u c h *)
END_IF


pChannel := ADR(CNCSystem.Channel[nChanIdx]);

(* Synch M-Functions *)
IF stTechnoAttributeData.nFunctionNumber_r > 0 AND stTechnoAttributeData.nFunctionNumber_r < 1000 THEN
	IF NOT pChannel^.M[stTechnoAttributeData.nFunctionNumber_r].bRes THEN					(* M-Function not set *)
		pChannel^.M[stTechnoAttributeData.nFunctionNumber_r].bState_rw				:= TRUE;	(* set M-Function *)
		pChannel^.M[stTechnoAttributeData.nFunctionNumber_r].nArgument_r		:= stTechnoAttributeData.nArgument_r;
		pChannel^.M[stTechnoAttributeData.nFunctionNumber_r].nBlockNumber_r		:= stTechnoAttributeData.nBlockNumber_r;
		pChannel^.M[stTechnoAttributeData.nFunctionNumber_r].nPrgLineNumber_r	:= stTechnoAttributeData.nPrgLineNumber_r;
		pChannel^.M[stTechnoAttributeData.nFunctionNumber_r].nFunctionNumber_r	:= stTechnoAttributeData.nFunctionNumber_r;
		pChannel^.M[stTechnoAttributeData.nFunctionNumber_r].nTime_r			:= stTechnoAttributeData.nTime_r;		
		pChannel^.M[stTechnoAttributeData.nFunctionNumber_r].bRes 				:= TRUE;	(* set acknowledge *)
		pChannel^.actM_r := CONCAT('M', UDINT_TO_STRING(stTechnoAttributeData.nFunctionNumber_r));
	ELSE
		IF NOT pChannel^.M[stTechnoAttributeData.nFunctionNumber_r].bState_rw THEN				(* wait for quit *)
			pChannel^.M[stTechnoAttributeData.nFunctionNumber_r].bRes 			:= FALSE;	(* quit the ack *)
			pChannel^.M[stTechnoAttributeData.nFunctionNumber_r].nArgument_r	:= 0;		(* reset the argument *)
			pChannel^.M[stTechnoAttributeData.nFunctionNumber_r].nBlockNumber_r		:= 0;
			pChannel^.M[stTechnoAttributeData.nFunctionNumber_r].nPrgLineNumber_r	:= 0;
			pChannel^.M[stTechnoAttributeData.nFunctionNumber_r].nFunctionNumber_r	:= 0;
			pChannel^.M[stTechnoAttributeData.nFunctionNumber_r].nTime_r			:= 0;				
			pChannel^.actM_r :='';
			bBusy 							:= FALSE;	(* quit *)
		END_IF
	END_IF
END_IF


(* Quit M00, M01, M02 , M17, M29, M30 *)
IF 	stTechnoAttributeData.nFunctionNumber_r = 0 OR 
	stTechnoAttributeData.nFunctionNumber_r = 01 OR 
	stTechnoAttributeData.nFunctionNumber_r = 02 OR 
	stTechnoAttributeData.nFunctionNumber_r = 17  OR 
	stTechnoAttributeData.nFunctionNumber_r = 29  OR 
	stTechnoAttributeData.nFunctionNumber_r = 30 THEN
		pChannel^.M[stTechnoAttributeData.nFunctionNumber_r].bState_rw 			:= FALSE;
		pChannel^.M[stTechnoAttributeData.nFunctionNumber_r].nArgument_r	:= 0;
		pChannel^.M[stTechnoAttributeData.nFunctionNumber_r].bRes 			:= FALSE;
		bBusy 							:= FALSE;
END_IF

END_FUNCTION_BLOCK

// ---- CNC Beckhoff/4 MHT-Function/HLI3_DoChannelTFunction.TcPOU
FUNCTION_BLOCK HLI3_DoChannelTFunction
VAR_INPUT
	/// Channel number 
	nChanIdx: INT;
	/// Number of T-function 
	nFuncNr: UDINT;
END_VAR
VAR_OUTPUT
	bBusy: BOOL;
END_VAR
VAR
	bStartTimer: BOOL;
END_VAR

(* ========================================================= *)
(*     FB: HLI_DoChannelTFunction                            *)
(* --------------------------------------------------------- *)
(*   Desc:                                                   *)
(* Author: MK, MiB                                           *)
(*   Rev.: 1.1                                               *)
(*   Date: 18.07.2002                                        *)
(*       : 08.04.2005, 03.03.2016 							 *)
(* ========================================================= *)


bBusy := FALSE;
RETURN;

IF NOT HLI3_CheckChannelValid(nChannel := nChanIdx) THEN
	RETURN; (* A b b r u c h *)
END_IF
bBusy := TRUE;

CASE nChanIdx OF
	0:	(* cnc channel 1 -------------------------------------- *)
		CASE nFuncNr OF
			0:		bBusy := FALSE;
			1:		bBusy := FALSE;
			2:		bBusy := FALSE;
			3:		bBusy := FALSE;
			4:		bBusy := FALSE;
			5:		bBusy := FALSE;
			6:		bBusy := FALSE;
			7:		bBusy := FALSE;
			8:		bBusy := FALSE;

			ELSE
			ADSLOGDINT( msgCtrlMask :=    ADSLOG_MSGTYPE_MSGBOX
			                           OR ADSLOG_MSGTYPE_LOG,
						msgFmtStr   := 'T-Funktion (%d), Channel 1, HLI_DoChannelTFunction() not implemented!',
						dintArg     := UDINT_TO_DINT(nFuncNr));
				(* Quit the M-Function *)
				bBusy := TRUE;
		END_CASE;


	1:	(* cnc channel 2 -------------------------------------- *)
		CASE nFuncNr OF
			0:		bBusy := FALSE;
			1:		bBusy := FALSE;
			2:		bBusy := FALSE;
			3:		bBusy := FALSE;


			ELSE
				ADSLOGDINT( msgCtrlMask :=    ADSLOG_MSGTYPE_MSGBOX
				                           OR ADSLOG_MSGTYPE_LOG,
							msgFmtStr   := 'T-Funktion (%d), Channel 2, HLI_DoChannelTFunction() not implemented!',
							dintArg     := UDINT_TO_DINT(nFuncNr));
				(* Quit the M-Function *)
				bBusy := FALSE;
		END_CASE;

ELSE
	ADSLOGDINT( msgCtrlMask :=    ADSLOG_MSGTYPE_MSGBOX
	                           OR ADSLOG_MSGTYPE_LOG,
				msgFmtStr   := 'Unknown channel number (%d) in HLI_DoChannelTFunction',
				dintArg     := INT_TO_DINT(nChanIdx));
	bBusy := FALSE;
END_CASE;

END_FUNCTION_BLOCK

// ---- CNC Beckhoff/4 MHT-Function/HLI3_DoChannelHFunction.TcPOU
FUNCTION_BLOCK HLI3_DoChannelHFunction
VAR_INPUT
	/// Channel number 
	nChanIdx: INT;
	stTechnoAttributeData: St_TechnoAttributeData;
END_VAR
VAR_OUTPUT
	bBusy: BOOL;
END_VAR
VAR
	pChannel: POINTER TO ST_CncChannel;
END_VAR

(* ========================================================= *)
(*     FB: HLI_DoChannelHFunction                            *)
(* --------------------------------------------------------- *)
(*   Desc:                                                   *)
(* Author: MiB                                               *)
(*   Rev.: 1.0                                               *)
(*   Date: 24.11.2010                                        *)
(*       : 08.04.2005                                        *)
(* ========================================================= *)
(* Rev.:	1.2												 *)
(* Date:	26.01.2011                                   	 *)
(* Author:	HR												 *)
(* Author:	Added support for additional h function number	 *)
(*			via new input variable 'nArg'				 	 *)
(* ========================================================= *)
bBusy := TRUE;

IF NOT HLI3_CheckChannelValid(nChannel := nChanIdx) THEN
	RETURN; (* A b b r u c h *)
END_IF


pChannel := ADR(CNCSystem.Channel[nChanIdx]);

(* Synch M-Functions *)
IF stTechnoAttributeData.nFunctionNumber_r > 0 AND stTechnoAttributeData.nFunctionNumber_r < 1000 THEN
	IF NOT pChannel^.H[stTechnoAttributeData.nFunctionNumber_r].bRes THEN					(* M-Function not set *)
		pChannel^.H[stTechnoAttributeData.nFunctionNumber_r].bState_rw				:= TRUE;	(* set M-Function *)
		pChannel^.H[stTechnoAttributeData.nFunctionNumber_r].nArgument_r		:= stTechnoAttributeData.nArgument_r;
		pChannel^.H[stTechnoAttributeData.nFunctionNumber_r].nBlockNumber_r		:= stTechnoAttributeData.nBlockNumber_r;
		pChannel^.H[stTechnoAttributeData.nFunctionNumber_r].nPrgLineNumber_r	:= stTechnoAttributeData.nPrgLineNumber_r;
		pChannel^.H[stTechnoAttributeData.nFunctionNumber_r].nFunctionNumber_r	:= stTechnoAttributeData.nFunctionNumber_r;
		pChannel^.H[stTechnoAttributeData.nFunctionNumber_r].nTime_r			:= stTechnoAttributeData.nTime_r;		
		pChannel^.H[stTechnoAttributeData.nFunctionNumber_r].bRes 				:= TRUE;	(* set acknowledge *)
		pChannel^.actH_r := CONCAT('H', UDINT_TO_STRING(stTechnoAttributeData.nFunctionNumber_r));
	ELSE
		IF NOT pChannel^.H[stTechnoAttributeData.nFunctionNumber_r].bState_rw THEN				(* wait for quit *)
			pChannel^.H[stTechnoAttributeData.nFunctionNumber_r].bRes 			:= FALSE;	(* quit the ack *)
			pChannel^.H[stTechnoAttributeData.nFunctionNumber_r].nArgument_r	:= 0;		(* reset the argument *)
			pChannel^.H[stTechnoAttributeData.nFunctionNumber_r].nBlockNumber_r		:= 0;
			pChannel^.H[stTechnoAttributeData.nFunctionNumber_r].nPrgLineNumber_r	:= 0;
			pChannel^.H[stTechnoAttributeData.nFunctionNumber_r].nFunctionNumber_r	:= 0;
			pChannel^.h[stTechnoAttributeData.nFunctionNumber_r].nTime_r			:= 0;
			pChannel^.actH_r := '';					
			bBusy 							:= FALSE;	(* quit *)
		END_IF
	END_IF
END_IF

END_FUNCTION_BLOCK

// ---- CNC Beckhoff/2 OperationMode/HLI3_ChannelResetRequest.TcPOU
FUNCTION_BLOCK HLI3_ChannelResetRequest
VAR_INPUT
	bExec: BOOL;
	/// Channel number 
	nChanIdx: INT;
	pChannel: POINTER TO ST_CncChannel;
END_VAR
VAR_OUTPUT
	bBusy: BOOL;
	bSwitchMode: BOOL;
	nMode: UDINT;
END_VAR
VAR
	fbRtrigExec: R_TRIG;
	/// Index of channel specific HLI area 
	nHliChIfcIdx: INT;
	nState: UINT;
	pCommand: POINTER TO HLI_PROC_TRANS_TO_MODE_STATE;
	actualMode: UDINT;
	fbTON: TON;
END_VAR

(******************************************************************************)
(* POU:				HLI_ChannelResetRequest									*)
(* Type:				Function block										*)
(* Customer:		Common													*)
(* Date:				07/11/16											*)
(* Last:				10/03/10											*)
(* -------------------------------------------------------------------------- *)
(* Revision:		1.0														*)
(* Author:			MiB														*)
(* Description: 	Performs a reset in the given cnc channel. 				*)
(* -------------------------------------------------------------------------- *)
(* Revision:		1.10													*)
(* Author:			MiB														*)
(* Description: 	Changed from PRG to FB.									*)
(* -------------------------------------------------------------------------- *)
(* Revision:		2.00															*)
(* Author:			HR																*)
(* Description: 	Deleted references to global variable 'PLCMachineMode[n]'.		*)
(*						The FB now works with VAR_OUTPUT 'nMode' and 'bSwitchMode'	*)
(*						as a callback to the initiator to let it perform the change	*)
(*						of the operation mode by itself in order to reset the cnc	*)
(*						channel.													*)
(* -------------------------------------------------------------------------- *)
(* Revision:		2.01																			*)
(* Author:			TV																				*)
(* Description: 	Expand State "Wait for previous mode"  *)
(*				Prevent to trigger the state machine during the mode switch							*)
(* -------------------------------------------------------------------------- *)
(* Revision:		2.02																			*)
(* Author:			MiB																				*)
(* Description: 	Tc3*)
(******************************************************************************)


fbRtrigExec( clk := bExec   );

IF fbRtrigExec.Q THEN
	bBusy := TRUE;
	nState := 10;
END_IF


CASE nState OF

0:		(* IDLE *)
		bBusy := FALSE;

10:	(* Reset request: get actual opmode *)
		bSwitchMode := FALSE;
		actualMode := gpCh[nChanIdx]^.channel_mc_control.mode_and_state.state_r.mode;
		nState := nState + 10;

20:  (* switch to standby *)
		bSwitchMode := TRUE;
		nMode:= HLI_IMCM_STANDBY_MODE;
		fbTON(IN:= FALSE);
		nState := nState + 10;

30: 	(* Wait for modeswitch *)
		bSwitchMode := FALSE;
		fbTON(IN:= TRUE, PT:= t#2000ms);
	 	IF gpCh[nChanIdx]^.channel_mc_control.mode_and_state.state_r.mode = HLI_IMCM_STANDBY_MODE THEN
			nState := nState + 10;
		END_IF
		IF fbTON.Q THEN
			(* Timeout Error -> go on with next step *)
			nState := nState + 10;
		END_IF

40:	(* switch back to previous mode *)
		bSwitchMode := TRUE;
		nMode:= actualMode;
		fbTON(IN:= FALSE);
		nState := nState + 10;

50:	(* Wait for previous mode  *)
		fbTON(IN:= TRUE, PT:= t#2000ms);
		IF (gpCh[nChanIdx]^.channel_mc_control.mode_and_state.state_r.mode = 	actualMode) THEN
			nState := nState + 10;
		END_IF
		IF fbTON.Q THEN
			(* Timeout Error -> go on with next step *)
			nState := nState + 10;
		END_IF

60: 	(* ready *)
		bSwitchMode := FALSE;
		nState := 0;

END_CASE



(* das muss ins aufrufende Programm: (HLI_CNCChannel)

VAR
	bResetRequest:			BOOL;
	fbRTrigReset:			R_TRIG;
	ChannelResetRequest: HLI_ChannelResetRequest;
END_VAR

fbRTrigReset(clk := bStateReset);
IF fbRTrigReset.Q THEN
	bResetRequest := TRUE;
	...
END_IF

(* Handle Channel reset *)
ChannelResetRequest
	(bExec 		:= bResetRequest ,
	 nChan 		:= nChan,
	 pChannel	:= ADR(CNCSystem.Channel[nChan])
	);

IF ChannelResetRequest.bSwitchMode THEN
	bModeStandby	:= bModeStandby OR (ChannelResetRequest.nMode = HLI_IMCM_STANDBY_MODE);
	bModeAutomatic	:= bModeAutomatic OR (ChannelResetRequest.nMode = HLI_IMCM_AUTOMATIC_MODE);
	bModeManual		:= bModeManual OR (ChannelResetRequest.nMode = HLI_IMCM_MANUAL_MODE);
	bModeMDI			:= bModeMDI OR (ChannelResetRequest.nMode = HLI_IMCM_MDI_MODE);
	bModeReference	:= bModeReference OR (ChannelResetRequest.nMode = HLI_IMCM_REFERENCE_MODE);
END_IF

IF bResetRequest AND NOT ChannelResetRequest.bBusy THEN
	bResetRequest := FALSE;
END_IF

*)

END_FUNCTION_BLOCK

// ---- CNC Beckhoff/3 Control/HLI3_ChannelSetBackwardMotion.TcPOU
FUNCTION HLI3_ChannelSetBackwardMotion : BOOL
VAR_INPUT
	/// Number of channel 
	nChanIdx: INT;
	bBackwardMotion: BOOL;
END_VAR

(* ========================================================= *)
(*    FUN: HLI_ChannelSetBackwardMotion                      *)
(* --------------------------------------------------------- *)
(*   Desc:                                                   *)
(* Author: MK, MiB                                           *)
(*   Date: 20.11.2012                                        *)
(*   Rev.: 1.1                                               *)
(* ========================================================= *)

HLI3_ChannelSetBackwardMotion := FALSE;
IF NOT HLI3_CheckChannelValid(nChannel := nChanIdx) THEN
	RETURN;
END_IF

gpCh[nChanIdx]^.bahn_mc_control.backward_motion.command_w := bBackwardMotion;

HLI3_ChannelSetBackwardMotion := TRUE;

END_FUNCTION

// ---- CNC Beckhoff/3 Control/HLI3_ChannelSetProgramBlockIgnore.TcPOU
FUNCTION HLI3_ChannelSetProgramBlockIgnore : BOOL
VAR_INPUT
	/// Number of channel 
	nChanIdx: INT;
	bPrgBlockIgnore: BOOL;
END_VAR

(* ========================================================= *)
(*    FUN: HLI_SetProgramBlockIgnore                         *)
(* --------------------------------------------------------- *)
(*   Desc:                                                   *)
(* Author: MK, MiB , TV                                      *)
(*   Date: 20.12.2012                                        *)
(*   Last: 19.11.2013                                        *)
(*   Rev.: 1.0                                               *)
(* ========================================================= *)

HLI3_ChannelSetProgramBlockIgnore := FALSE;
IF NOT HLI3_CheckChannelValid(nChannel := nChanIdx) THEN
	RETURN;
END_IF

(* program block ignore *)
IF bPrgBlockIgnore THEN
	gpCh[nChanIdx]^.decoder_mc_control.program_block_ignore.command_w := 1;
ELSE
	gpCh[nChanIdx]^.decoder_mc_control.program_block_ignore.command_w := 0;
END_IF

HLI3_ChannelSetProgramBlockIgnore := TRUE;

END_FUNCTION

// ---- CNC Beckhoff/3 Control/HLI3_ChannelSetFeedHold.TcPOU
FUNCTION HLI3_ChannelSetFeedHold : BOOL
VAR_INPUT
	/// Number of channel 
	nChanIdx: INT;
	bFeedHold: BOOL;
END_VAR

(* ========================================================= *)
(*    FUN: HLI_ChannelSetFeedHold                            *)
(* --------------------------------------------------------- *)
(*   Desc:                                                   *)
(* Author: MK , MiB                                          *)
(*   Date: 20.11.2012                                        *)
(*   Rev.: 1.1                                               *)
(* ========================================================= *)

HLI3_ChannelSetFeedHold := FALSE;
IF NOT HLI3_CheckChannelValid(nChannel := nChanIdx) THEN
	RETURN;
END_IF

(* if the stop button from the HMI is selected the request is set *)
gpCh[nChanIdx]^.bahn_mc_control.feedhold.command_w := bFeedHold OR gpCh[nChanIdx]^.bahn_mc_control.feedhold.request_r;
HLI3_ChannelSetFeedHold := TRUE;

END_FUNCTION

// ---- CNC Beckhoff/3 Control/HLI3_ChannelSetSingleBlock.TcPOU
FUNCTION HLI3_ChannelSetSingleBlock : BOOL
VAR_INPUT
	/// Number of channel 
	nChanIdx: INT;
	bSingleBlock: BOOL;
END_VAR

(* ========================================================= *)
(*    FUN: HLI3_ChannelSetSingleBlock                        *)
(* --------------------------------------------------------- *)
(*   Desc:                                                   *)
(* Author: MK ,MiB                                           *)
(*   Date: 20.11.2012                                        *)
(*   Rev.: 1.1                                               *)
(* ========================================================= *)

HLI3_ChannelSetSingleBlock := FALSE;
IF NOT HLI3_CheckChannelValid(nChannel := nChanIdx) THEN
	RETURN;
END_IF
gpCh[nChanIdx]^.bahn_mc_control.single_block.command_w   := bSingleBlock;

HLI3_ChannelSetSingleBlock := TRUE;

END_FUNCTION

// ---- CNC Beckhoff/3 Control/HLI3_ChannelSetReducedFeed.TcPOU
FUNCTION HLI3_ChannelSetReducedFeed : BOOL
VAR_INPUT
	/// Number of channel 
	nChanIdx: INT;
	bReducedFeed: BOOL;
END_VAR

(* ========================================================= *)
(*    FUN: HLI_ChannelSetReducedFeed                         *)
(* --------------------------------------------------------- *)
(*   Desc:                                                   *)
(* Author: MK,MiB                                            *)
(*   Date: 20.11.2012                                        *)
(*   Rev.: 1.1                                               *)
(* ========================================================= *)


HLI3_ChannelSetReducedFeed := FALSE;
IF NOT HLI3_CheckChannelValid(nChannel := nChanIdx) THEN
	RETURN;
END_IF
gpCh[nChanIdx]^.bahn_mc_control.reduced_speed.command_w := bReducedFeed;
HLI3_ChannelSetReducedFeed := TRUE;

END_FUNCTION

// ---- CNC Beckhoff/4 MHT-Function/HLI3_ChannelResetMFunctions.TcPOU
FUNCTION HLI3_ChannelResetMFunctions : BOOL
VAR_INPUT
	/// Channel number 
	nChanIdx: INT;
END_VAR
VAR
	idx: INT;
END_VAR

(* ========================================================= *)
(*    FUN: HLI_ChannelResetMFunctions                        *)
(* --------------------------------------------------------- *)
(*   Desc:                                                   *)
(* Author: MK                                                *)
(*   Date: 10.05.2007                                        *)
(*   Rev.: 1.00                                              *)
(* ========================================================= *)

IF NOT HLI3_CheckChannelValid(nChannel := nChanIdx) THEN
	HLI3_ChannelResetMFunctions := FALSE;
	RETURN; (* A b b r u c h *)
END_IF


FOR idx := 1 TO 999 DO
	CNCSystem.Channel[nChanIdx].M[idx].bState_rw := FALSE;
	CNCSystem.Channel[nChanIdx].M[idx].bRes := FALSE;
	CNCSystem.Channel[nChanIdx].actM_r :='';
END_FOR

HLI3_ChannelResetMFunctions := TRUE;

END_FUNCTION

// ---- CNC Beckhoff/4 MHT-Function/HLI3_ChannelResetHFunctions.TcPOU
FUNCTION HLI3_ChannelResetHFunctions : BOOL
VAR_INPUT
	/// Channel number 
	nChanIdx: INT;
END_VAR
VAR
	idx: INT;
END_VAR

(* ========================================================= *)
(*    FUN: HLI_ChannelResetHFunctions                        *)
(* --------------------------------------------------------- *)
(*   Desc:                                                   *)
(* Author: MiB                                                *)
(*   Date: 23.11.2012                                        *)
(*   Rev.: 1.1                                              *)
(* ========================================================= *)



IF NOT HLI3_CheckChannelValid(nChannel := nChanIdx) THEN
	HLI3_ChannelResetHFunctions := FALSE;
	RETURN; (* A b b r u c h *)
END_IF


FOR idx := 0 TO 999 DO
	CNCSystem.Channel[nChanIdx].H[idx].bState_rw := FALSE;
	CNCSystem.Channel[nChanIdx].H[idx].bRes := FALSE;
	CNCSystem.Channel[nChanIdx].actH_r :='';
END_FOR

HLI3_ChannelResetHFunctions := TRUE;

END_FUNCTION

// ---- CNC Beckhoff/3 Control/HLI3_GetChannelStatusInfo.TcPOU
FUNCTION HLI3_GetChannelStatusInfo : BOOL
VAR_INPUT
	/// Number of channel 
	nChanIdx: INT;
END_VAR
VAR
	pChannel: POINTER TO ST_CNCChannel;
END_VAR

(* ========================================================= *)
(*    FUN: HLI_GetStatusInfo                                 *)
(* --------------------------------------------------------- *)
(*   Desc: Status Info from the HLI Interface                *)
(* Author: MK,Mib                                            *)
(*   Date: 18.07.2002                                        *)
(*   Rev.: 1.0                                               *)
(* ========================================================= *)

IF NOT HLI3_CheckChannelValid(nChannel := nChanIdx) THEN
	RETURN;
END_IF


pChannel := ADR(CNCSystem.Channel[nChanIdx]);
pChannel^.ActMode := HLI3_GetChannelMode(nChanIdx:=nChanIdx);
pChannel^.ActState := HLI3_GetChannelState(nChanIdx:=nChanIdx);



(* Translate mode *)
CASE pChannel^.ActMode OF
	HLI_IMCM_MODE:					pChannel^.ActModeString := 'Mode';
	HLI_IMCM_STANDBY_MODE:			pChannel^.ActModeString := 'StandbyMode';
	HLI_IMCM_AUTOMATIC_MODE:		pChannel^.ActModeString := 'AutomaticMode';
	HLI_IMCM_MDI_MODE:				pChannel^.ActModeString := 'MDIMode';
	HLI_IMCM_MANUAL_MODE:			pChannel^.ActModeString := 'ManualMode';
	HLI_IMCM_REFERENCE_MODE:		pChannel^.ActModeString := 'ReferenceMode';
ELSE
	pChannel^.ActModeString := '---';
END_CASE;

(* Translate state *)
CASE pChannel^.ActState OF
	HLI_IMCM_PROCESS_DESELECTED:	pChannel^.ActStateString := 'Deselected';
	HLI_IMCM_PROCESS_SELECTED:		pChannel^.ActStateString := 'Selected';
	HLI_IMCM_PROCESS_READY:			pChannel^.ActStateString := 'Ready';
	HLI_IMCM_PROCESS_ACTIVE:		pChannel^.ActStateString := 'Active';
	HLI_IMCM_PROCESS_HOLD:			pChannel^.ActStateString := 'Hold';
	HLI_IMCM_PROCESS_ERROR:			pChannel^.ActStateString := 'Error';
	HLI_IMCM_PROCESS_SELECTING:		pChannel^.ActStateString := 'Selecting';
	HLI_IMCM_PROCESS_DESELECTING:	pChannel^.ActStateString := 'Deselecting';
	HLI_IMCM_PROCESS_PREPARING:		pChannel^.ActStateString := 'Preparing';
	HLI_IMCM_PROCESS_CLEARING:		pChannel^.ActStateString := 'Clearing';
	HLI_IMCM_PROCESS_STARTING:		pChannel^.ActStateString := 'Starting';
	HLI_IMCM_PROCESS_ABORTING:		pChannel^.ActStateString := 'Aborting';
	HLI_IMCM_PROCESS_STOPPING:		pChannel^.ActStateString := 'Stopping';
	HLI_IMCM_PROCESS_RESUMING:		pChannel^.ActStateString := 'Resuming';
	HLI_IMCM_PROCESS_RESETTING:		pChannel^.ActStateString := 'Resetting';
	HLI_IMCM_PROCESS_FINISHING:		pChannel^.ActStateString := 'Finishing';
ELSE
	pChannel^.ActStateString := '---';
END_CASE;

END_FUNCTION

// ---- CNC Beckhoff/3 Control/HLI3_GetChannelMode.TcPOU
FUNCTION HLI3_GetChannelMode : UDINT
VAR_INPUT
	/// Number of channel 
	nChanIdx: INT;
END_VAR

(* ========================================================= *)
(*    FUN: HLI_GetChannelMode                                *)
(* --------------------------------------------------------- *)
(*   Desc:                                                   *)
(* Author: MK                                                *)
(*   Date: 18.07.2002                                        *)
(*   Rev.: 1.0                                               *)
(* ========================================================= *)
HLI3_GetChannelMode := 0;
IF NOT HLI3_CheckChannelValid(nChannel := nChanIdx) THEN
	RETURN;
END_IF

(* if the stop button from the HMI is selected the request is set *)
HLI3_GetChannelMode := gpCh[nChanIdx]^.channel_mc_control.mode_and_state.state_r.mode;

END_FUNCTION

// ---- CNC Beckhoff/3 Control/HLI3_GetChannelState.TcPOU
FUNCTION HLI3_GetChannelState : UDINT
VAR_INPUT
	/// Number of channel 
	nChanIdx: INT;
END_VAR

(* ========================================================= *)
(*    FUN: HLI3_GetChannelState                              *)
(* --------------------------------------------------------- *)
(*   Desc:                                                   *)
(* Author: MK                                                *)
(*   Date: 18.07.2002                                        *)
(*   Rev.: 1.0                                               *)
(* ========================================================= *)

HLI3_GetChannelState := 0;
IF NOT HLI3_CheckChannelValid(nChannel := nChanIdx) THEN
	RETURN;
END_IF

(* if the stop button from the HMI is selected the request is set *)
HLI3_GetChannelState := gpCh[nChanIdx]^.channel_mc_control.mode_and_state.state_r.state;

END_FUNCTION

// ---- CNC Beckhoff/3 Control/HLI3_GetChannelError.TcPOU
FUNCTION HLI3_GetChannelError : BOOL
VAR_INPUT
	/// Number of channel 
	nChanIdx: INT;
END_VAR
VAR
	pChannel: POINTER TO ST_CNCChannel;
END_VAR

(* ========================================================= *)
(*    FUN: HLI_GetChannelError                               *)
(* --------------------------------------------------------- *)
(*   Desc: Gets the channel error                            *)
(* Return: The error flag of the channel                     *)
(* Author: MK , MiB, TV                                      *)
(*   Date: 08.07.2015                                        *)
(*   Rev.: 1.3                                               *)
(* ========================================================= *)

IF NOT HLI3_CheckChannelValid(nChannel := nChanIdx) THEN
	RETURN;
END_IF

pChannel := ADR(CNCSystem.Channel[nChanIdx]);

(* Visualisation of Mode and State *)
pChannel^.ActMode  := HLI3_GetChannelMode(nChanIdx:=nChanIdx);
pChannel^.ActState := HLI3_GetChannelState(nChanIdx:=nChanIdx);

(* Error messages id *)
IF pChannel^.ActState = HLI_IMCM_PROCESS_ERROR THEN
	pChannel^.Error := TRUE;	
ELSE
	pChannel^.Error := FALSE;	
END_IF

END_FUNCTION

// ---- CNC Beckhoff/2 OperationMode/HLI3_ChannelModeStandby.TcPOU
FUNCTION HLI3_ChannelModeStandby : BOOL
VAR_INPUT	 
	ProgramName: STRING(HLI_IMCM_MODE_STATE_PARAM_STRL);
	pUnit: POINTER TO MC_CONTROL_MCM_MODE_STATE_UNIT;
	pCommand: POINTER TO HLI_PROC_TRANS_TO_MODE_STATE;
	pChannel: POINTER TO ST_CncChannel;
END_VAR
VAR
	pString: POINTER TO STRING(HLI_IMCM_MODE_STATE_PARAM_STRL);
END_VAR

(* ========================================================= *)
(*    FUN: HLI_ChannelModeStandby                            *)
(* --------------------------------------------------------- *)
(*   Desc: switch channel to Standby mode / xxx              *)
(* Author: MK, MiB, TV                                       *)
(*   Date: 02.07.2015                                        *)
(*   Rev.: 1.2                                              *)
(* ========================================================= *)

IF (NOT pUnit^.command_semaphor_rw) THEN  (* only if semaphor is FALSE...... *)
	IF pChannel^.State.Selected THEN
		pChannel^.State.Selected := FALSE;
		pCommand^.to_mode := HLI_IMCM_STANDBY_MODE;
		pCommand^.to_state := HLI_IMCM_PROCESS_SELECTED;		
		pString := ADR(pCommand^.parameter);
		pString^ := ProgramName;
		pUnit^.command_semaphor_rw := TRUE;
		ADSLOG(strMsg:='Standby Mode selected', nDINT:=0, strArg := '');
	END_IF
	
	IF pChannel^.State.Ready THEN
		pChannel^.State.Ready := FALSE;
		pCommand^.to_mode := HLI_IMCM_STANDBY_MODE;
		pCommand^.to_state := HLI_IMCM_PROCESS_READY;		
		pString := ADR(pCommand^.parameter);
		pString^ := ProgramName;
		pUnit^.command_semaphor_rw := TRUE;
		ADSLOG(strMsg:='Standby Mode ready', nDINT:=0, strArg := '');
	END_IF
	
	IF pChannel^.State.Start THEN
		pChannel^.State.Start := FALSE;
		pCommand^.to_mode := HLI_IMCM_STANDBY_MODE;
		pCommand^.to_state := HLI_IMCM_PROCESS_ACTIVE;		
		pString := ADR(pCommand^.parameter);
		pString^ := ProgramName;
		pUnit^.command_semaphor_rw := TRUE;
		ADSLOG(strMsg:='Programm %s started', nDINT:=0, strArg:=ProgramName);
	END_IF
	
	IF pChannel^.State.Stop THEN
		pChannel^.State.Stop := FALSE;
		pCommand^.to_mode := HLI_IMCM_STANDBY_MODE;
		pCommand^.to_state := HLI_IMCM_PROCESS_HOLD;		
		pUnit^.command_semaphor_rw := TRUE;
		ADSLOG(strMsg:='Standby Mode stopped', nDINT:=0, strArg := '');
	END_IF
	
	IF pChannel^.State.Reset THEN
		pChannel^.State.Reset := FALSE;
		pCommand^.to_mode := HLI_IMCM_STANDBY_MODE;
		pCommand^.to_state := HLI_IMCM_PROCESS_DESELECTED;		
		pUnit^.command_semaphor_rw := TRUE;
		ADSLOG(strMsg:='Standby Mode resetting', nDINT:=0, strArg := '');
	END_IF
	
	HLI3_ChannelModeStandby := TRUE;
ELSE
	HLI3_ChannelModeStandby := FALSE;
END_IF

END_FUNCTION

// ---- CNC Beckhoff/2 OperationMode/HLI3_ChannelModeAuto.TcPOU
FUNCTION HLI3_ChannelModeAuto : BOOL
VAR_INPUT	
	ProgramName: STRING(HLI_IMCM_MODE_STATE_PARAM_STRL);
	pUnit: POINTER TO MC_CONTROL_MCM_MODE_STATE_UNIT;
	pCommand: POINTER TO HLI_PROC_TRANS_TO_MODE_STATE;
	pChannel: POINTER TO ST_CncChannel;
END_VAR
VAR
	pString: POINTER TO STRING(HLI_IMCM_MODE_STATE_PARAM_STRL);
END_VAR

(* ========================================================= *)
(*    FUN: HLI_ChannelModeAuto                               *)
(* --------------------------------------------------------- *)
(*   Desc: switch channel to Automatic mode / xxx            *)
(* Author: MK,MiB, TV                                        *)
(*   Date: 19.08.2015                                        *)
(*   Rev.: 1.3                                               *)
(* ========================================================= *)

IF (NOT pUnit^.command_semaphor_rw) THEN    (* only if semaphor is FALSE...... *)
	IF pChannel^.State.Selected THEN
		pChannel^.State.Selected := FALSE;
		pCommand^.to_mode := HLI_IMCM_AUTOMATIC_MODE;
		pCommand^.to_state := HLI_IMCM_PROCESS_SELECTED;	
		pString := ADR(pCommand^.parameter);
		pString^ := ProgramName;
		pUnit^.command_semaphor_rw := TRUE;
		ADSLOG(strMsg:='Automatic selected', nDINT:=0, strArg := '');
	END_IF
	
	IF pChannel^.State.Ready THEN
		pChannel^.State.Ready := FALSE;
		pCommand^.to_mode := HLI_IMCM_AUTOMATIC_MODE;
		pCommand^.to_state := HLI_IMCM_PROCESS_READY;		
		pString := ADR(pCommand^.parameter);
		pString^ := ProgramName;
		pUnit^.command_semaphor_rw := TRUE;
		ADSLOG(strMsg:='Automatic ready', nDINT:=0, strArg := '');
	END_IF
	
	IF pChannel^.State.Start THEN
		pChannel^.State.Start := FALSE;
		pCommand^.to_mode := HLI_IMCM_AUTOMATIC_MODE;
		pCommand^.to_state := HLI_IMCM_PROCESS_ACTIVE;		
		pString := ADR(pCommand^.parameter);
		pString^ := ProgramName;
		pUnit^.command_semaphor_rw := TRUE;
		ADSLOG(strMsg:='Programm %s started', nDINT:=0, strArg:=ProgramName);
	END_IF
	
	IF pChannel^.State.Stop THEN
		pChannel^.State.Stop := FALSE;
		pCommand^.to_mode := HLI_IMCM_AUTOMATIC_MODE;
		pCommand^.to_state := HLI_IMCM_PROCESS_HOLD;		
		pUnit^.command_semaphor_rw := TRUE;
		ADSLOG(strMsg:='Programm stopped', nDINT:=0, strArg := '');
	END_IF
	
	IF pChannel^.State.Reset THEN
		pChannel^.State.Reset := FALSE;
		pCommand^.to_mode := HLI_IMCM_AUTOMATIC_MODE;
		pCommand^.to_state := HLI_IMCM_PROCESS_RESETTING;		
		pUnit^.command_semaphor_rw := TRUE;
		ADSLOG(strMsg:='Automatic resetting', nDINT:=0, strArg := '');
	END_IF
	
	HLI3_ChannelModeAuto := TRUE;
ELSE
	HLI3_ChannelModeAuto := FALSE;
END_IF

END_FUNCTION

// ---- CNC Beckhoff/2 OperationMode/HLI3_ChannelModeMDI.TcPOU
FUNCTION HLI3_ChannelModeMDI : BOOL
VAR_INPUT	
	/// pointer to the MDI program string 
	pMDIString: POINTER TO STRING(HLI_IMCM_MODE_STATE_PARAM_STRL);
	pUnit: POINTER TO MC_CONTROL_MCM_MODE_STATE_UNIT;
	pCommand: POINTER TO HLI_PROC_TRANS_TO_MODE_STATE;
	pChannel: POINTER TO ST_CncChannel;
END_VAR
VAR
	pString: POINTER TO STRING(HLI_IMCM_MODE_STATE_PARAM_STRL);
END_VAR

(* ========================================================= *)
(*    FUN: HLI_ChannelModeMDI                                *)
(* --------------------------------------------------------- *)
(*   Desc: switch channel to MDI mode / xxx                  *)
(*   Author: MK, TV, MiB, Rch                                *)
(*   Date: 18.07.2002                                        *)
(*   Last: 19.08.2015                      				     *)
(*   Rev.: 1.5                                               *)
(* ========================================================= *)

IF (NOT pUnit^.command_semaphor_rw) THEN  (* only if semaphor is FALSE...... *)

	IF pChannel^.State.Selected THEN
		pChannel^.State.Selected := FALSE;
		pCommand^.to_mode := HLI_IMCM_MDI_MODE;
		pCommand^.to_state := HLI_IMCM_PROCESS_SELECTED;		
		pString := ADR(pCommand^.parameter);
		pString^ := pMDIString^;
		pUnit^.command_semaphor_rw := TRUE;
		ADSLOG(strMsg:='MDI Mode selected', nDINT:=0, strArg := '');
	END_IF
	
	IF pChannel^.State.Ready THEN
		pChannel^.State.Ready := FALSE;
		pCommand^.to_mode := HLI_IMCM_MDI_MODE;
		pCommand^.to_state := HLI_IMCM_PROCESS_READY;		
		pUnit^.command_semaphor_rw := TRUE;
		ADSLOG(strMsg:='MDI Mode ready', nDINT:=0, strArg := '');
	END_IF
	
	IF pChannel^.State.Start THEN
		pChannel^.State.Start := FALSE;
		pCommand^.to_mode := HLI_IMCM_MDI_MODE;
		pCommand^.to_state := HLI_IMCM_PROCESS_ACTIVE;
		pString := ADR(pCommand^.parameter);
		pString^ := pMDIString^;
		pUnit^.command_semaphor_rw := TRUE;
		ADSLOG(strMsg:='MDI %s started', nDINT:=0, strArg:=pMDIString^);
	END_IF
	
	IF pChannel^.State.Stop THEN
		pChannel^.State.Stop := FALSE;
		pCommand^.to_mode := HLI_IMCM_MDI_MODE;
		pCommand^.to_state := HLI_IMCM_PROCESS_HOLD;		
		pUnit^.command_semaphor_rw := TRUE;
		ADSLOG(strMsg:='MDI Mode stopped', nDINT:=0, strArg := '');
	END_IF
	
	IF pChannel^.State.Reset THEN
		pChannel^.State.Reset := FALSE;
		pCommand^.to_mode := HLI_IMCM_MDI_MODE;
		pCommand^.to_state := HLI_IMCM_PROCESS_RESETTING;		
		pUnit^.command_semaphor_rw := TRUE;
		ADSLOG(strMsg:='MDI Mode resetting', nDINT:=0, strArg := '');
	END_IF
	HLI3_ChannelModeMDI := TRUE;	
ELSE
	HLI3_ChannelModeMDI := FALSE;
END_IF

END_FUNCTION

// ---- CNC Beckhoff/2 OperationMode/HLI3_ChannelModeReference.TcPOU
FUNCTION HLI3_ChannelModeReference : BOOL
VAR_INPUT	
	/// the referencing string 
	sRefPosString: STRING(HLI_IMCM_MODE_STATE_PARAM_STRL);
	pUnit: POINTER TO MC_CONTROL_MCM_MODE_STATE_UNIT;
	pCommand: POINTER TO HLI_PROC_TRANS_TO_MODE_STATE;
	pChannel: POINTER TO ST_CncChannel;
END_VAR
VAR
	pString: POINTER TO STRING(HLI_IMCM_MODE_STATE_PARAM_STRL);
END_VAR

(* ========================================================= *)
(*    FUN: HLI_ChannelModeReference                          *)
(* --------------------------------------------------------- *)
(*   Desc: switch channel to Reference mode / xxx            *)
(* Author: MK, MiB, TV                                       *)
(*   Date: 02.07.2015                                        *)
(*   Rev.: 1.3                                               *)
(* ========================================================= *)


(************************************************************
	RefPosString:
	Element: parameter ( ASCII char set, Länge:256 Zeichen)

	Vorgabe zur Parametrierung der Referenzpunktfahrt.

	Ist dieser STRING leer, so wird defaultmäßig das
	Automatikprogramm "rpf.nc" angewählt.

	Ansonsten kann durch explizite Angabe der Achsen und
	Zeitpunkt im Format "G74
	<Achsbezeichner_1><Zeitpunkt_1> ...
	<Achsbezeichner_n><Zeitpunkt_n>"
	eine individuelle Referenzpunktfahrt vorgegeben werden.
*************************************************************)

IF (NOT pUnit^.command_semaphor_rw) THEN  (* only if semaphor is FALSE...... *)
	IF pChannel^.State.Selected THEN
		pChannel^.State.Selected := FALSE;
		pCommand^.to_mode := HLI_IMCM_REFERENCE_MODE;
		pCommand^.to_state := HLI_IMCM_PROCESS_SELECTED;		
		pUnit^.command_semaphor_rw := TRUE;
		ADSLOG(strMsg:='Reference selected', nDINT:=0, strArg:='');
	END_IF
	
	IF pChannel^.State.Ready THEN
		pChannel^.State.Ready := FALSE;
		pCommand^.to_mode := HLI_IMCM_REFERENCE_MODE;
		pCommand^.to_state := HLI_IMCM_PROCESS_READY;		
		pString := ADR(pCommand^.parameter);
		pUnit^.command_semaphor_rw := TRUE;
		ADSLOG(strMsg:='MDI Mode ready', nDINT:=0, strArg := '');
	END_IF
	
	IF pChannel^.State.Start THEN
		pChannel^.State.Start := FALSE;
		pCommand^.to_mode := HLI_IMCM_REFERENCE_MODE;
		pCommand^.to_state := HLI_IMCM_PROCESS_ACTIVE;		
		pString := ADR(pCommand^.parameter);
		pString^ := sRefPosString;
		pUnit^.command_semaphor_rw := TRUE;
		ADSLOG(strMsg:='Programm %s reference is started', nDINT:=0, strArg:=sRefPosString);
	END_IF
	
	IF pChannel^.State.Stop THEN
		pChannel^.State.Stop := FALSE;
		pCommand^.to_mode := HLI_IMCM_REFERENCE_MODE;
		pCommand^.to_state := HLI_IMCM_PROCESS_HOLD;		
		pUnit^.command_semaphor_rw := TRUE;
		ADSLOG(strMsg:='Reference stop is selected', nDINT:=0, strArg:='');
	END_IF
	
	IF pChannel^.State.Reset THEN
		pChannel^.State.Reset := FALSE;
		pCommand^.to_mode := HLI_IMCM_REFERENCE_MODE;
		pCommand^.to_state := HLI_IMCM_PROCESS_DESELECTED;		
		pUnit^.command_semaphor_rw := TRUE;
		ADSLOG(strMsg:='Reference reset is selected', nDINT:=0, strArg:='');
	END_IF

	HLI3_ChannelModeReference := TRUE;
ELSE
	HLI3_ChannelModeReference := FALSE;
END_IF

END_FUNCTION

// ---- CNC Beckhoff/2 OperationMode/HLI3_ChannelModeManual.TcPOU
FUNCTION HLI3_ChannelModeManual : BOOL
VAR_INPUT	
	pUnit: POINTER TO MC_CONTROL_MCM_MODE_STATE_UNIT;
	pCommand: POINTER TO HLI_PROC_TRANS_TO_MODE_STATE;
	pChannel: POINTER TO ST_CncChannel;
	sManualInitString : STRING;
END_VAR
VAR
	pString: POINTER TO STRING;
END_VAR

(* ========================================================= *)
(*    FUN: HLI_ChannelModeManual                             *)
(* --------------------------------------------------------- *)
(*   Desc: switch channel to Manual mode / xxx               *)
(* Author: MK, MiB, TV, RCH                                  *)
(*   Date: 19.08.2015                                        *)
(*   Rev.: 1.2                                               *)
(* ========================================================= *)

IF (NOT pUnit^.command_semaphor_rw) THEN    (* only if semaphor is FALSE...... *)
	IF pChannel^.State.Selected THEN
		pChannel^.State.Selected := FALSE;
		pCommand^.to_mode := HLI_IMCM_MANUAL_MODE;
		pCommand^.to_state := HLI_IMCM_PROCESS_SELECTED;		
		pString := ADR(pCommand^.parameter);
		pString^ := '';
		pUnit^.command_semaphor_rw := TRUE;
		ADSLOG(strMsg:='Manual Mode selected', nDINT:=0, strArg := '');
	END_IF
	
	IF pChannel^.State.Ready THEN
		pChannel^.State.Ready := FALSE;
		pCommand^.to_mode := HLI_IMCM_MANUAL_MODE;
		pCommand^.to_state := HLI_IMCM_PROCESS_READY;		
		pString := ADR(pCommand^.parameter);
		pString^ := '';
		pUnit^.command_semaphor_rw := TRUE;
		ADSLOG(strMsg:='Manual Mode ready', nDINT:=0, strArg := '');
	END_IF
	
	IF pChannel^.State.Start THEN
		pChannel^.State.Start := FALSE;
		pCommand^.to_mode := HLI_IMCM_MANUAL_MODE;
		pCommand^.to_state := HLI_IMCM_PROCESS_ACTIVE;		
		pString := ADR(pCommand^.parameter);
        pString^ := sManualInitString;								(* Unterprogramm zur Initialisierung des Handbetriebes *)
		pUnit^.command_semaphor_rw := TRUE;
		ADSLOG(strMsg:='Manual Mode active', nDINT:=0, strArg := '');
	END_IF
	
	IF pChannel^.State.Stop THEN
		pChannel^.State.Stop := FALSE;
		pCommand^.to_mode := HLI_IMCM_MANUAL_MODE;
		pCommand^.to_state := HLI_IMCM_PROCESS_HOLD;		
		pUnit^.command_semaphor_rw := TRUE;
		ADSLOG(strMsg:='Manual Mode stopped', nDINT:=0, strArg := '');
	END_IF
	
	IF pChannel^.State.Reset THEN
		pChannel^.State.Reset := FALSE;
		pCommand^.to_mode := HLI_IMCM_MANUAL_MODE;
		pCommand^.to_state := HLI_IMCM_PROCESS_RESETTING;		
		pUnit^.command_semaphor_rw := TRUE;
		ADSLOG(strMsg:='Manual Mode resetting', nDINT:=0, strArg := '');
	END_IF

	HLI3_ChannelModeManual := TRUE;
ELSE
	HLI3_ChannelModeManual := FALSE;
END_IF

END_FUNCTION

// ---- CNC Beckhoff/2 OperationMode/HLI3_ChannelReset.TcPOU
FUNCTION HLI3_ChannelReset : BOOL
VAR_INPUT
	/// Channel index 
	nChanIdx: INT;
END_VAR
VAR
	/// local pointer to Data of actual Channel 
	pChannelData: POINTER TO HIGH_LEVEL_INTERFACE_CH;
END_VAR

(* ========================================================= *)
(*    FUN: HLI_ChannelReset                                  *)
(* --------------------------------------------------------- *)
(*   Desc:                                                   *)
(* Author: MK ,MiB                                           *)
(*   Date: 20.11.2012                                        *)
(*   Rev.: 1.1                                               *)
(* ========================================================= *)


HLI3_ChannelReset := FALSE;
IF NOT HLI3_CheckChannelValid(nChannel := nChanIdx) THEN
	RETURN;
END_IF

(* get pointer to channel data *)
pChannelData := gpCh[nChanIdx];
IF (pChannelData = 0) THEN   (* check for zero pointer *)
	RETURN;
END_IF

(* is a reset commanded *)
IF pChannelData^.bahn_lc_control.plc_reset.command_r = TRUE THEN
	(* quit this reset *)
	pChannelData^.bahn_lc_control.plc_reset.state_w := TRUE;
	ADSLOG(strMsg:='Reset of channel: %d', nDINT:=INT_TO_DINT(nChanIdx), strArg:='');
	HLI3_ChannelReset := TRUE;
END_IF

END_FUNCTION

// ---- CNC Beckhoff/2 OperationMode/HLI3_AxisReset.TcPOU
FUNCTION HLI3_AxisReset : BOOL
VAR_INPUT
	/// Channel number 
	nChanNo: INT;
	/// Axis number 
	nHliAxisIdx: INT;
END_VAR
VAR
	/// local pointer to data of actual axis 
	pAxisData: POINTER TO HIGH_LEVEL_INTERFACE_AX;
END_VAR

(* ========================================================= *)
(*    FUN: HLI3_QuitAxisReset                                 *)
(* --------------------------------------------------------- *)
(*   Desc:                                                   *)
(* Author: MK , MiB                                          *)
(*   Date: 20.11.2012                                        *)
(*   Rev.: 1.1                                               *)
(* ========================================================= *)


HLI3_AxisReset := FALSE;
IF NOT HLI3_CheckAxisValid(nHliAxisIdx := nHliAxisIdx) THEN
	RETURN;
END_IF

IF gpAx[nHliAxisIdx] = 0 THEN
	RETURN;
END_IF


(* get pointer to axis data *)
pAxisData := gpAx[nHliAxisIdx];
IF pAxisData^.ipo_state.cnc_channel_r = INT_TO_UINT(nChanNo) THEN (* it's an axis of the channel *)
	(* is a reset commanded *)
	IF pAxisData^.ipo_lc_control.plc_reset.command_r = TRUE THEN
		(* quit this reset *)
		pAxisData^.ipo_lc_control.plc_reset.state_w := TRUE;

		ADSLOG(strMsg:='Reset of axis: %d', nDINT:=INT_TO_DINT(nHliAxisIdx), strArg:='');

		HLI3_AxisReset := TRUE;
	END_IF
END_IF

END_FUNCTION

// ---- CNC Beckhoff/6 BlockSearch/HLI3_BlockSearch.TcPOU
FUNCTION_BLOCK HLI3_BlockSearch
VAR_INPUT
	/// Number of channel 
	nChanIdx: INT;
	/// interface values 
	BlockSearch: ST_BlockSearch;
END_VAR
VAR_IN_OUT
	/// Edge signal 
	bStartWrite: BOOL;
	/// Edge signal 
	bStartRead: BOOL;
END_VAR
VAR_OUTPUT
	Busy: BOOL;
	Err: BOOL;
	nErrorState: UINT;
	/// interface values 
	nActType: INT;
	fActDistance: LREAL;
	bActAutoReturn: BOOL;
	nActDeviationMax: UDINT;
	nActBlockNumber: DINT;
	nActPass: DINT;
	nActBlockCount: DINT;
	/// current values 
	actualBlockNumber: DINT := 0;
	actualBlockCount: UDINT := 0;
	actualBlockCount_AfterReset: UDINT := 0;
	coveredDistance: DINT;
	coveredDistance_AfterReset: DINT := 0;
END_VAR
VAR
	bReadStarted: BOOL;
	bWriteStarted: BOOL;
	rtStartRead: R_TRIG;
	rtStartWrite: R_TRIG;
	writeType: WriteBsType;
	readType: ReadBsType;
	writeDistance: WriteBsCoveredDistance;
	readDistance: ReadBsCoveredDistance;
	writeAutoReturn: WriteBsAutoReturn;
	readAutoReturn: ReadBsAutoReturn;
	writeDeviationMax: WriteBsDeviationMax;
	readDeviationMax: ReadBsDeviationMax;
	writeBlockNumber: WriteBsBlockNumber;
	ReadBlockNumber: ReadBsBlockNumber;
	writeBlockCount: WriteBsBlockCount;
	ReadBlockCount: ReadBsBlockCount;	
	writePass: WriteBsPass;
	readPass: ReadBsPass;
	nChannelIdxGrp: UDINT;
	/// Timer to read axisposition cyclically        
	Timer: TON;
	actualcoveredDistance: BOOL;
	ChannelMode: UDINT;
	BlockSearchStart: BOOL;
END_VAR

(* ---------------------*----------------------------------|------------------------------------------------------- *)
(* PURPOSE:                                                                                                         *)
(*                                                                                                                  *)
(*                                                                                                                  *)
(* SCOPE:                                                                                                           *)
(*                                                                                                                  *)
(*                                                                                                                  *)
(* REMARKS:                                                                                                         *)
(*                                                                                                                  *)
(*                                                                                                                  *)
(* AUTHOR:              VERSION     DATE                   CHECKED FROM      DATE     STATUS                        *)
(*    MK                1.0         07.05.2003                                                                      *)
(*    TV                1.1         10.06.2006                                                                      *)
(*    TV                1.2         20.08.2014                                                                      *)
(*    TV                1.2         29.09.2014                                                                      *)
(*    TV                1.3         25.06.2015                                                                      *)
(* ---------------------*----------------------------------|------------------------------------------------------- *)

IF NOT HLI3_CheckChannelValid(nChannel := nChanIdx) THEN
	RETURN;
END_IF




Err := FALSE;
nChannelIdxGrp := 16#00020100 + INT_TO_UDINT(nChanIdx)+1;
BlockSearchStart := FALSE;


(* ----------------------------------- *)
(* --- write block search commands --- *)
(* ----------------------------------- *)

rtStartWrite(CLK:=bStartWrite);
IF rtStartWrite.Q THEN
   bWriteStarted := TRUE;
   bStartWrite := FALSE; (* reset the HMI signal *)
END_IF

IF bWriteStarted THEN
   Busy := TRUE;
   IF BlockSearch.nType = 5 THEN
   	BlockSearch.nType := 3;								(* start position by block count *)

		BlockSearch.bAutoReturn := TRUE;
		(*nPass	:= 1;*)
	END_IF

	(* write block search data to memory *)
   writeType(nIdxGrp:=nChannelIdxGrp, bStart:=rtStartWrite.Q, nType:=BlockSearch.nType);
   writeDistance(nIdxGrp:=nChannelIdxGrp, bStart:=rtStartWrite.Q, fDistance:=(BlockSearch.fDistance*10.0));
   writeAutoReturn(nIdxGrp:=nChannelIdxGrp, bStart:=rtStartWrite.Q, bAutoReturn:=BlockSearch.bAutoReturn);
   writeDeviationMax(nIdxGrp:=nChannelIdxGrp, bStart:=rtStartWrite.Q, nDeviationMax:=BlockSearch.nDeviationMax);
   writePass(nIdxGrp:=nChannelIdxGrp, bStart:=rtStartWrite.Q, nPass:=BlockSearch.nPass);

	CASE BlockSearch.nType OF		(* count and number share a part of the memory *)
		3: writeBlockCount(nIdxGrp:=nChannelIdxGrp, bStart:=rtStartWrite.Q, nBlockCount:=BlockSearch.nBlockCount);
		4: writeBlockNumber(nIdxGrp:=nChannelIdxGrp, bStart:=rtStartWrite.Q, nBlockNumber:=BlockSearch.nBlockNumber);
   END_CASE

   IF writeType.Busy = FALSE
      AND writeDistance.BUSY = FALSE
      AND writeAutoReturn.BUSY = FALSE
      AND writeDeviationMax.BUSY = FALSE
      AND writeBlockNumber.BUSY = FALSE
      AND writePass.BUSY = FALSE
      AND writeBlockCount.BUSY = FALSE
   THEN
      Busy := FALSE;
      bWriteStarted := FALSE;
      BlockSearchStart := TRUE;
   END_IF
END_IF


(* Satzsuchlauf starten *)

(*
IF (BlockSearchStart) AND ((nType = 3) OR (nType = 4)) THEN
	PLCMachineMode[nChan].Start := TRUE;
END_IF
*)

(* -------------------------------- *)
(* --- read block search states --- *)
(* -------------------------------- *)

(* the next rows only for test *)
(* Start a cyclic timer with period 2 sec. *)
Timer(IN := NOT(Timer.Q), PT := T#2000ms);

rtStartRead(CLK:=bStartRead);
(*rtStartRead(CLK:=Timer.Q);*)
IF rtStartRead.Q THEN
   bReadStarted := TRUE;
END_IF

IF bReadStarted THEN
	Busy := TRUE;

   readType(nIdxGrp:=nChannelIdxGrp, bStart:=rtStartRead.Q, pDest:=ADR(nActType));
   readDistance(nIdxGrp:=nChannelIdxGrp, bStart:=rtStartRead.Q, pDest:=ADR(fActDistance));
   readAutoReturn(nIdxGrp:=nChannelIdxGrp, bStart:=rtStartRead.Q, pDest:=ADR(bActAutoReturn));
   readDeviationMax(nIdxGrp:=nChannelIdxGrp, bStart:=rtStartRead.Q, pDest:=ADR(nActDeviationMax));
	CASE nActType OF			(* count and number cannot be read within a single cycle! *)
		3: readBlockCount(nIdxGrp:=nChannelIdxGrp, bStart:=rtStartRead.Q, pDest:=ADR(nActBlockCount));
		4: readBlockNumber(nIdxGrp:=nChannelIdxGrp, bStart:=rtStartRead.Q, pDest:=ADR(nActBlockNumber));
	END_CASE;
   readPass(nIdxGrp:=nChannelIdxGrp, bStart:=rtStartRead.Q, pDest:=ADR(nActPass));

   (*
   readActualBlockNumber(nIdxGrp:=nChannelIdxGrp, bStart:=rtStartRead.Q, pDest:=ADR(actualBlockNumber));
   readActualBlockCount(nIdxGrp:=nChannelIdxGrp, bStart:=rtStartRead.Q, pDest:=ADR(actualBlockCount));
   *)

   IF readType.Busy = FALSE
      AND readDistance.Busy = FALSE
      AND readAutoReturn.Busy = FALSE
      AND readDeviationMax.Busy = FALSE
      AND readBlockNumber.Busy = FALSE
      AND readPass.Busy = FALSE      
   THEN
		Busy := FALSE;

		bReadStarted := FALSE;
		bStartRead := FALSE; (* reset the HMI signal *)
   END_IF
END_IF

actualBlockNumber := gpCh[nChanIdx]^.bahn_state.block_nr_r;
actualBlockCount  := gpCh[nChanIdx]^.bahn_state.block_count_r; 

coveredDistance := gpCh[nChanIdx]^.bahn_state.covered_distance_r;  (* just read actual covered distance *)

(* Speichert die Unterbrechungsstelle *)
ChannelMode := HLI3_GetChannelMode(nChanIdx);
IF (actualBlockCount <> 0) AND (ChannelMode = 2) AND (CNCSystem.Channel[nChanIdx].ActState =4) THEN
	actualBlockCount_AfterReset := actualBlockCount;									(* Zeiger bleibt auch nach Reset erhalten *)
	coveredDistance_AfterReset := coveredDistance;
END_IF

(*	UnterbrechungsstelleWeg			:= coveredDistance/10.0;*)

(*actualBlockNumber := gpAx[0]^.lr_state.block_nr_r;  asume first axis is always moved *)


(* handshake during block search on/off *)
gpCh[nChanIdx]^.bahn_lc_control.block_search.enable_w := TRUE;

IF gpCh[nChanIdx]^.bahn_lc_control.block_search.command_r <>
   gpCh[nChanIdx]^.bahn_lc_control.block_search.state_w THEN

   (* acknowledge *)
   gpCh[nChanIdx]^.bahn_lc_control.block_search.state_w :=
      gpCh[nChanIdx]^.bahn_lc_control.block_search.command_r;

(*
   (* pup up of change *)
   IF gpCh[nHliChIfcIdx]^.bahn_lc_control.block_search.state_w THEN
      ADSLOGDINT( msgCtrlMask := ADSLOG_MSGTYPE_MSGBOX OR ADSLOG_MSGTYPE_LOG,
                  msgFmtStr := 'block search: %d', dintArg := 1);
   ELSE
      ADSLOGDINT( msgCtrlMask := ADSLOG_MSGTYPE_MSGBOX OR ADSLOG_MSGTYPE_LOG,
                  msgFmtStr := 'block search: %d', dintArg := 0);
   END_IF
*)
END_IF

END_FUNCTION_BLOCK

// ---- CNC Beckhoff/6 BlockSearch/WriteBsType.TcPOU
FUNCTION_BLOCK WriteBsType
VAR_INPUT
	nIdxGrp: UDINT;
	bStart: BOOL;
	nType: UINT;
END_VAR
VAR_OUTPUT
	Busy: BOOL;
	bErr: BOOL;
END_VAR
VAR
	fbWrite: ADSWRITE;
	bStarted: BOOL;
END_VAR

IF bStarted = FALSE THEN
   IF bStart = TRUE THEN
      bStarted := TRUE;
      bErr := FALSE;
      Busy := TRUE;
   END_IF
END_IF

IF bStarted THEN
   (* raising edge of Timer triggers write request *)
   fbWrite( NetID := '', Port := 553, IdxGrp := nIdxGrp, IdxOffs := 16#00000049,
         LEN := 2, SrcAddr := ADR(nType), WRITE := bStarted, TMOUT := T#1s);
   IF NOT fbWrite.Busy THEN
      (* There was an error in the execution of the write request *)
      IF fbWrite.Err THEN
         bErr := TRUE;
      END_IF
      fbWrite(WRITE := FALSE);    (* reset because of edge detection in FB ADSWRITE *)
      bStarted := FALSE;
      Busy := FALSE;
   END_IF
END_IF

END_FUNCTION_BLOCK

// ---- CNC Beckhoff/6 BlockSearch/ReadBsType.TcPOU
FUNCTION_BLOCK ReadBsType
VAR_INPUT
	nIdxGrp: UDINT;
	bStart: BOOL;
	pDest: POINTER TO UINT;
END_VAR
VAR_OUTPUT
	Busy: BOOL;
	bErr: BOOL;
END_VAR
VAR
	fbRead: ADSREAD;
	bStarted: BOOL;
END_VAR

IF bStarted = FALSE THEN
   IF bStart = TRUE THEN
      bStarted := TRUE;
      bErr := FALSE;
      Busy := TRUE;
   END_IF
END_IF

IF bStarted THEN
   (* raising edge of Timer triggers read request *)
   fbRead( NetID := '', Port := 553, IdxGrp := nIdxGrp, IdxOffs := 16#00000061,
         LEN := 2, DestAddr := pDest, READ := bStarted, TMOUT := T#1s);
   IF NOT fbRead.Busy THEN
      (* There was an error in the execution of the read request *)
      IF fbRead.Err THEN
         bErr := TRUE;
      END_IF
      fbRead(READ := FALSE);    (* reset because of edge detection in FB ADSREAD *)
      bStarted := FALSE;
      Busy := FALSE;
   END_IF
END_IF

END_FUNCTION_BLOCK

// ---- CNC Beckhoff/6 BlockSearch/WriteBsCoveredDistance.TcPOU
FUNCTION_BLOCK WriteBsCoveredDistance
VAR_INPUT
	nIdxGrp: UDINT;
	bStart: BOOL;
	fDistance: LREAL;
END_VAR
VAR_OUTPUT
	Busy: BOOL;
	bErr: BOOL;
END_VAR
VAR
	fbWrite: ADSWRITE;
	bStarted: BOOL;
END_VAR

IF bStarted = FALSE THEN
   IF bStart = TRUE THEN
      bStarted := TRUE;
      bErr := FALSE;
      Busy := TRUE;
   END_IF
END_IF

IF bStarted THEN
   (* raising edge of Timer triggers write request *)
   fbWrite( NetID := '', Port := 553, IdxGrp := nIdxGrp, IdxOffs := 16#0000004A,
         LEN := 8, SrcAddr := ADR(fDistance), WRITE := bStarted, TMOUT := T#1s);
   IF NOT fbWrite.Busy THEN
      (* There was an error in the execution of the write request *)
      IF fbWrite.Err THEN
         bErr := TRUE;
      END_IF
      fbWrite(WRITE := FALSE);    (* reset because of edge detection in FB ADSWRITE *)
      bStarted := FALSE;
      Busy := FALSE;
   END_IF
END_IF

END_FUNCTION_BLOCK

// ---- CNC Beckhoff/6 BlockSearch/ReadBsCoveredDistance.TcPOU
FUNCTION_BLOCK ReadBsCoveredDistance
VAR_INPUT
	nIdxGrp: UDINT;
	bStart: BOOL;
	pDest: POINTER TO LREAL;
END_VAR
VAR_OUTPUT
	Busy: BOOL;
	bErr: BOOL;
END_VAR
VAR
	fbRead: ADSREAD;
	bStarted: BOOL;
END_VAR

IF bStarted = FALSE THEN
   IF bStart = TRUE THEN
      bStarted := TRUE;
      bErr := FALSE;
      Busy := TRUE;
   END_IF
END_IF

IF bStarted THEN
   (* raising edge of Timer triggers read request *)
   fbRead( NetID := '', Port := 553, IdxGrp := nIdxGrp, IdxOffs := 16#00000062,
         LEN := 8, DestAddr := pDest, READ := bStarted, TMOUT := T#1s);
   IF NOT fbRead.Busy THEN
      (* There was an error in the execution of the read request *)
      IF fbRead.Err THEN
         bErr := TRUE;
      END_IF
      fbRead(READ := FALSE);    (* reset because of edge detection in FB ADSREAD *)
      bStarted := FALSE;
      Busy := FALSE;
   END_IF
END_IF

END_FUNCTION_BLOCK

// ---- CNC Beckhoff/6 BlockSearch/WriteBsAutoReturn.TcPOU
FUNCTION_BLOCK WriteBsAutoReturn
VAR_INPUT
	nIdxGrp: UDINT;
	bStart: BOOL;
	bAutoReturn: BOOL;
END_VAR
VAR_OUTPUT
	Busy: BOOL;
	bErr: BOOL;
END_VAR
VAR
	fbWrite: ADSWRITE;
	bStarted: BOOL;
END_VAR

IF bStarted = FALSE THEN
   IF bStart = TRUE THEN
      bStarted := TRUE;
      bErr := FALSE;
      Busy := TRUE;
   END_IF
END_IF

IF bStarted THEN
   (* raising edge of Timer triggers write request *)
   fbWrite( NetID := '', Port := 553, IdxGrp := nIdxGrp, IdxOffs := 16#0000004B,
         LEN := 1, SrcAddr := ADR(bAutoReturn), WRITE := bStarted, TMOUT := T#1s);
   IF NOT fbWrite.Busy THEN
      (* There was an error in the execution of the write request *)
      IF fbWrite.Err THEN
         bErr := TRUE;
      END_IF
      fbWrite(WRITE := FALSE);    (* reset because of edge detection in FB ADSWRITE *)
      bStarted := FALSE;
      Busy := FALSE;
   END_IF
END_IF

END_FUNCTION_BLOCK

// ---- CNC Beckhoff/6 BlockSearch/ReadBsAutoReturn.TcPOU
FUNCTION_BLOCK ReadBsAutoReturn
VAR_INPUT
	nIdxGrp: UDINT;
	bStart: BOOL;
	pDest: POINTER TO BOOL;
END_VAR
VAR_OUTPUT
	Busy: BOOL;
	bErr: BOOL;
END_VAR
VAR
	fbRead: ADSREAD;
	bStarted: BOOL;
END_VAR

IF bStarted = FALSE THEN
   IF bStart = TRUE THEN
      bStarted := TRUE;
      bErr := FALSE;
      Busy := TRUE;
   END_IF
END_IF

IF bStarted THEN
   (* raising edge of Timer triggers read request *)
   fbRead( NetID := '', Port := 553, IdxGrp := nIdxGrp, IdxOffs := 16#00000063,
         LEN := 1, DestAddr := pDest, READ := bStarted, TMOUT := T#1s);
   IF NOT fbRead.Busy THEN
      (* There was an error in the execution of the read request *)
      IF fbRead.Err THEN
         bErr := TRUE;
      END_IF
      fbRead(READ := FALSE);    (* reset because of edge detection in FB ADSREAD *)
      bStarted := FALSE;
      Busy := FALSE;
   END_IF
END_IF

END_FUNCTION_BLOCK

// ---- CNC Beckhoff/6 BlockSearch/WriteBsDeviationMax.TcPOU
FUNCTION_BLOCK WriteBsDeviationMax
VAR_INPUT
	nIdxGrp: UDINT;
	bStart: BOOL;
	nDeviationMax: UDINT;
END_VAR
VAR_OUTPUT
	Busy: BOOL;
	bErr: BOOL;
END_VAR
VAR
	fbWrite: ADSWRITE;
	bStarted: BOOL;
END_VAR

IF bStarted = FALSE THEN
   IF bStart = TRUE THEN
      bStarted := TRUE;
      bErr := FALSE;
      Busy := TRUE;
   END_IF
END_IF

IF bStarted THEN
   (* raising edge of Timer triggers write request *)
   fbWrite( NetID := '', Port := 553, IdxGrp := nIdxGrp, IdxOffs := 16#0000004C,
         LEN := 4, SrcAddr := ADR(nDeviationMax), WRITE := bStarted, TMOUT := T#1s);
   IF NOT fbWrite.Busy THEN
      (* There was an error in the execution of the write request *)
      IF fbWrite.Err THEN
         bErr := TRUE;
      END_IF
      fbWrite(WRITE := FALSE);    (* reset because of edge detection in FB ADSWRITE *)
      bStarted := FALSE;
      Busy := FALSE;
   END_IF
END_IF

END_FUNCTION_BLOCK

// ---- CNC Beckhoff/6 BlockSearch/ReadBsDeviationMax.TcPOU
FUNCTION_BLOCK ReadBsDeviationMax
VAR_INPUT
	nIdxGrp: UDINT;
	bStart: BOOL;
	pDest: POINTER TO UDINT;
END_VAR
VAR_OUTPUT
	Busy: BOOL;
	bErr: BOOL;
END_VAR
VAR
	fbRead: ADSREAD;
	bStarted: BOOL;
END_VAR

IF bStarted = FALSE THEN
   IF bStart = TRUE THEN
      bStarted := TRUE;
      bErr := FALSE;
      Busy := TRUE;
   END_IF
END_IF

IF bStarted THEN
   (* raising edge of Timer triggers read request *)
   fbRead( NetID := '', Port := 553, IdxGrp := nIdxGrp, IdxOffs := 16#00000064,
         LEN := 4, DestAddr := pDest, READ := bStarted, TMOUT := T#1s);
   IF NOT fbRead.Busy THEN
      (* There was an error in the execution of the read request *)
      IF fbRead.Err THEN
         bErr := TRUE;
      END_IF
      fbRead(READ := FALSE);    (* reset because of edge detection in FB ADSREAD *)
      bStarted := FALSE;
      Busy := FALSE;
   END_IF
END_IF

END_FUNCTION_BLOCK

// ---- CNC Beckhoff/6 BlockSearch/WriteBsBlockNumber.TcPOU
FUNCTION_BLOCK WriteBsBlockNumber
VAR_INPUT
	nIdxGrp: UDINT;
	bStart: BOOL;
	nBlockNumber: DINT;
END_VAR
VAR_OUTPUT
	Busy: BOOL;
	bErr: BOOL;
END_VAR
VAR
	fbWrite: ADSWRITE;
	bStarted: BOOL;
END_VAR

IF bStarted = FALSE THEN
   IF bStart = TRUE THEN
      bStarted := TRUE;
      bErr := FALSE;
      Busy := TRUE;
   END_IF
END_IF

IF bStarted THEN
   (* raising edge of Timer triggers write request *)
   fbWrite( NetID := '', Port := 553, IdxGrp := nIdxGrp, IdxOffs := 16#0000005F,
         LEN := 4, SrcAddr := ADR(nBlockNumber), WRITE := bStarted, TMOUT := T#1s);
   IF NOT fbWrite.Busy THEN
      (* There was an error in the execution of the write request *)
      IF fbWrite.Err THEN
         bErr := TRUE;
      END_IF
      fbWrite(WRITE := FALSE);    (* reset because of edge detection in FB ADSWRITE *)
      bStarted := FALSE;
      Busy := FALSE;
   END_IF
END_IF

END_FUNCTION_BLOCK

// ---- CNC Beckhoff/6 BlockSearch/ReadBlockNumber.TcPOU
FUNCTION_BLOCK ReadBlockNumber
VAR_INPUT
	nIdxGrp: UDINT;
	bStart: BOOL;
	pDest: POINTER TO DINT;
END_VAR
VAR_OUTPUT
	Busy: BOOL;
	bErr: BOOL;
END_VAR
VAR
	fbRead: ADSREAD;
	bStarted: BOOL;
END_VAR

IF bStarted = FALSE THEN
   IF bStart = TRUE THEN
      bStarted := TRUE;
      bErr := FALSE;
      Busy := TRUE;
   END_IF
END_IF

IF bStarted THEN
   (* raising edge of Timer triggers read request *)
   fbRead( NetID := '', Port := 553, IdxGrp := nIdxGrp, IdxOffs := 16#0000000E,
         LEN := 4, DestAddr := pDest, READ := bStarted, TMOUT := T#1s);
   IF NOT fbRead.Busy THEN
      (* There was an error in the execution of the read request *)
      IF fbRead.Err THEN
         bErr := TRUE;
      END_IF
      fbRead(READ := FALSE);    (* reset because of edge detection in FB ADSREAD *)
      bStarted := FALSE;
      Busy := FALSE;
   END_IF
END_IF

END_FUNCTION_BLOCK

